LIN {X 0,Y 190.635,Z 472.728,A -85,B 0,C 180,E1 -21841.367,E2 -21841.367} C_VEL
LIN {X 0,Y 190.155,Z 472.929,A -85,B 0,C 180,E1 -21843.676,E2 -21843.676} C_VEL
LIN {X 0,Y 189.683,Z 472.071,A -85,B 0,C 180,E1 -21847.835,E2 -21847.835} C_VEL
LIN {X 0,Y 189.629,Z 470.742,A -85,B 0,C 180,E1 -21850.519,E2 -21850.519} C_VEL
LIN {X 0,Y 190.011,Z 467.936,A -85,B 0,C 180,E1 -21854.047,E2 -21854.047} C_VEL
LIN {X 0,Y 190.59,Z 464.351,A -85,B 0,C 180,E1 -21857.221,E2 -21857.221} C_VEL
LIN {X 0,Y 191.538,Z 459.248,A -85,B 0,C 180,E1 -21860.606,E2 -21860.606} C_VEL
LIN {X 0,Y 192.941,Z 452.066,A -85,B 0,C 180,E1 -21864.254,E2 -21864.254} C_VEL
LIN {X 0,Y 194.673,Z 443.985,A -85,B 0,C 180,E1 -21867.417,E2 -21867.417} C_VEL
LIN {X 0,Y 196.751,Z 434.772,A -85,B 0,C 180,E1 -21870.26,E2 -21870.26} C_VEL
LIN {X 0,Y 199.045,Z 424.398,A -85,B 0,C 180,E1 -21872.786,E2 -21872.786} C_VEL
LIN {X 0,Y 201.339,Z 412.61,A -85,B 0,C 180,E1 -21875.009,E2 -21875.009} C_VEL
LIN {X 0,Y 203.246,Z 401.02,A -85,B 0,C 180,E1 -21876.705,E2 -21876.705} C_VEL
LIN {X 0,Y 205.015,Z 388.044,A -85,B 0,C 180,E1 -21878.097,E2 -21878.097} C_VEL
LIN {X 0,Y 206.329,Z 374.818,A -85,B 0,C 180,E1 -21879.087,E2 -21879.087} C_VEL
LIN {X 0,Y 207.163,Z 361.086,A -85,B 0,C 180,E1 -21879.699,E2 -21879.699} C_VEL
LIN {X 0,Y 209.379,Z 305.404,A -85,B 0,C 180,E1 -21881.576,E2 -21881.576} C_VEL
LIN {X 0,Y 204.012,Z 288.584,A -85,B 0,C 180,E1 -21882.979,E2 -21882.979} C_VEL
LIN {X 0,Y 197.083,Z 272.096,A -85,B 0,C 180,E1 -21884.701,E2 -21884.701} C_VEL
LIN {X 0,Y 192.993,Z 264.168,A -85,B 0,C 180,E1 -21885.75,E2 -21885.75} C_VEL
LIN {X 0,Y 192.766,Z 263.116,A -85,B 0,C 180,E1 -21886.145,E2 -21886.145} C_VEL
LIN {X 0,Y 192.66,Z 262.98,A -85,B 0,C 180,E1 -21889.169,E2 -21889.169} C_VEL
LIN {X 0,Y 192.599,Z 262.997,A -85,B 0,C 180,E1 -21894.206,E2 -21894.206} C_VEL
LIN {X 0,Y 192.575,Z 263.001,A -85,B 0,C 180,E1 -21898.872,E2 -21898.872} C_VEL
LIN {X 0,Y 192.571,Z 262.983,A -85,B 0,C 180,E1 -21903.195,E2 -21903.195} C_VEL
LIN {X 0,Y 192.521,Z 262.988,A -85,B 0,C 180,E1 -21908.363,E2 -21908.363} C_VEL
LIN {X 0,Y 192.467,Z 263.009,A -85,B 0,C 180,E1 -21913.102,E2 -21913.102} C_VEL
LIN {X 0,Y 192.468,Z 262.995,A -85,B 0,C 180,E1 -21916.916,E2 -21916.916} C_VEL
LIN {X 0,Y 192.528,Z 262.99,A -85,B 0,C 180,E1 -21921.655,E2 -21921.655} C_VEL
LIN {X 0,Y 192.585,Z 262.985,A -85,B 0,C 180,E1 -21926.823,E2 -21926.823} C_VEL
LIN {X 0,Y 192.604,Z 262.959,A -85,B 0,C 180,E1 -21931.693,E2 -21931.693} C_VEL
LIN {X 0,Y 192.652,Z 262.986,A -85,B 0,C 180,E1 -21936.351,E2 -21936.351} C_VEL
LIN {X 0,Y 192.694,Z 262.947,A -85,B 0,C 180,E1 -21941.501,E2 -21941.501} C_VEL
LIN {X 0,Y 192.74,Z 262.946,A -85,B 0,C 180,E1 -21945.221,E2 -21945.221} C_VEL
LIN {X 0,Y 192.95,Z 262.949,A -85,B 0,C 180,E1 -21949.576,E2 -21949.576} C_VEL
LIN {X 0,Y 192.97,Z 262.926,A -85,B 0,C 180,E1 -21953.736,E2 -21953.736} C_VEL
LIN {X 0,Y 193.236,Z 262.875,A -85,B 0,C 180,E1 -21957.924,E2 -21957.924} C_VEL
LIN {X 0,Y 193.422,Z 262.875,A -85,B 0,C 180,E1 -21960.008,E2 -21960.008} C_VEL
LIN {X 0,Y 192.939,Z 262.951,A -85,B 0,C 180,E1 -21964.186,E2 -21964.186} C_VEL
LIN {X 0,Y 193.031,Z 262.904,A -85,B 0,C 180,E1 -21968.382,E2 -21968.382} C_VEL
LIN {X 0,Y 192.803,Z 262.955,A -85,B 0,C 180,E1 -21972.641,E2 -21972.641} C_VEL
LIN {X 0,Y 192.732,Z 262.972,A -85,B 0,C 180,E1 -21976.969,E2 -21976.969} C_VEL
LIN {X 0,Y 192.6,Z 262.967,A -85,B 0,C 180,E1 -21981.409,E2 -21981.409} C_VEL
LIN {X 0,Y 192.654,Z 262.984,A -85,B 0,C 180,E1 -21984.21,E2 -21984.21} C_VEL
LIN {X 0,Y 192.621,Z 262.97,A -85,B 0,C 180,E1 -21988.87,E2 -21988.87} C_VEL
LIN {X 0,Y 192.615,Z 262.993,A -85,B 0,C 180,E1 -21993.191,E2 -21993.191} C_VEL
LIN {X 0,Y 192.561,Z 262.99,A -85,B 0,C 180,E1 -21998.358,E2 -21998.358} C_VEL
LIN {X 0,Y 192.504,Z 262.993,A -85,B 0,C 180,E1 -22003.095,E2 -22003.095} C_VEL
LIN {X 0,Y 192.505,Z 262.996,A -85,B 0,C 180,E1 -22006.909,E2 -22006.909} C_VEL
LIN {X 0,Y 192.606,Z 263.152,A -85,B 0,C 180,E1 -22011.508,E2 -22011.508} C_VEL
LIN {X 0,Y 193.472,Z 266.43,A -85,B 0,C 180,E1 -22013.217,E2 -22013.217} C_VEL
LIN {X 0,Y 197.352,Z 275.633,A -85,B 0,C 180,E1 -22014.326,E2 -22014.326} C_VEL
LIN {X 0,Y 203.854,Z 292.087,A -85,B 0,C 180,E1 -22015.975,E2 -22015.975} C_VEL
LIN {X 0,Y 207.069,Z 301.489,A -85,B 0,C 180,E1 -22016.795,E2 -22016.795} C_VEL
LIN {X 0,Y 209.011,Z 318.594,A -85,B 0,C 180,E1 -22017.718,E2 -22017.718} C_VEL
LIN {X 0,Y 208.6,Z 329.617,A -85,B 0,C 180,E1 -22018.092,E2 -22018.092} C_VEL
LIN {X 0,Y 207.75,Z 335.448,A -85,B 0,C 180,E1 -22018.209,E2 -22018.209} C_VEL
LIN {X 0,Y 201.752,Z 354.354,A -85,B 0,C 180,E1 -22018.18,E2 -22018.18} C_VEL
LIN {X 0,Y 200.903,Z 360.185,A -85,B 0,C 180,E1 -22018.303,E2 -22018.303} C_VEL
LIN {X 0,Y 199.95,Z 377.377,A -85,B 0,C 180,E1 -22018.989,E2 -22018.989} C_VEL
LIN {X 0,Y 198.707,Z 390.244,A -85,B 0,C 180,E1 -22019.878,E2 -22019.878} C_VEL
LIN {X 0,Y 196.959,Z 403.1,A -85,B 0,C 180,E1 -22021.199,E2 -22021.199} C_VEL
LIN {X 0,Y 194.713,Z 415.331,A -85,B 0,C 180,E1 -22022.887,E2 -22022.887} C_VEL
LIN {X 0,Y 192.54,Z 426.271,A -85,B 0,C 180,E1 -22024.888,E2 -22024.888} C_VEL
LIN {X 0,Y 190.296,Z 437.059,A -85,B 0,C 180,E1 -22027.429,E2 -22027.429} C_VEL
LIN {X 0,Y 188.057,Z 446.823,A -85,B 0,C 180,E1 -22030.342,E2 -22030.342} C_VEL
LIN {X 0,Y 186.11,Z 455.204,A -85,B 0,C 180,E1 -22033.544,E2 -22033.544} C_VEL
LIN {X 0,Y 184.681,Z 461.939,A -85,B 0,C 180,E1 -22036.798,E2 -22036.798} C_VEL
LIN {X 0,Y 183.755,Z 467.292,A -85,B 0,C 180,E1 -22040.086,E2 -22040.086} C_VEL
LIN {X 0,Y 183.23,Z 471.435,A -85,B 0,C 180,E1 -22043.389,E2 -22043.389} C_VEL
LIN {X 0,Y 183.008,Z 474.694,A -85,B 0,C 180,E1 -22046.943,E2 -22046.943} C_VEL
LIN {X 0,Y 183.091,Z 476.56,A -85,B 0,C 180,E1 -22049.997,E2 -22049.997} C_VEL
LIN {X 0,Y 182.987,Z 477.614,A -85,B 0,C 180,E1 -22052.932,E2 -22052.932} C_VEL
LIN {X 0,Y 183.318,Z 477.942,A -85,B 0,C 180,E1 -22056.601,E2 -22056.601} C_VEL
LIN {X 0,Y 184.259,Z 476.916,A -85,B 0,C 180,E1 -22060.991,E2 -22060.991} C_VEL
LIN {X 0,Y 185.09,Z 475.826,A -85,B 0,C 180,E1 -22063.165,E2 -22063.165} C_VEL
LIN {X 0,Y 187.406,Z 472.371,A -85,B 0,C 180,E1 -22067.455,E2 -22067.455} C_VEL
LIN {X 0,Y 189.98,Z 468.647,A -85,B 0,C 180,E1 -22070.572,E2 -22070.572} C_VEL
LIN {X 0,Y 193.063,Z 463.838,A -85,B 0,C 180,E1 -22073.601,E2 -22073.601} C_VEL
LIN {X 0,Y 196.79,Z 457.336,A -85,B 0,C 180,E1 -22076.756,E2 -22076.756} C_VEL
LIN {X 0,Y 200.573,Z 450.34,A -85,B 0,C 180,E1 -22079.373,E2 -22079.373} C_VEL
LIN {X 0,Y 204.416,Z 442.725,A -85,B 0,C 180,E1 -22081.618,E2 -22081.618} C_VEL
LIN {X 0,Y 208.897,Z 432.451,A -85,B 0,C 180,E1 -22084.005,E2 -22084.005} C_VEL
LIN {X 0,Y 212.902,Z 422.02,A -85,B 0,C 180,E1 -22085.865,E2 -22085.865} C_VEL
LIN {X 0,Y 216.718,Z 410.439,A -85,B 0,C 180,E1 -22087.444,E2 -22087.444} C_VEL
LIN {X 0,Y 219.89,Z 398.149,A -85,B 0,C 180,E1 -22088.696,E2 -22088.696} C_VEL
LIN {X 0,Y 222.444,Z 385.35,A -85,B 0,C 180,E1 -22089.619,E2 -22089.619} C_VEL
LIN {X 0,Y 224.08,Z 373.434,A -85,B 0,C 180,E1 -22090.191,E2 -22090.191} C_VEL
LIN {X 0,Y 226.848,Z 330.995,A -85,B 0,C 180,E1 -22091.536,E2 -22091.536} C_VEL
LIN {X 0,Y 221.284,Z 318.167,A -85,B 0,C 180,E1 -22093.904,E2 -22093.904} C_VEL
LIN {X 0,Y 216.569,Z 309.026,A -85,B 0,C 180,E1 -22096.018,E2 -22096.018} C_VEL
LIN {X 0,Y 211.954,Z 300.85,A -85,B 0,C 180,E1 -22098.281,E2 -22098.281} C_VEL
LIN {X 0,Y 207.464,Z 293.64,A -85,B 0,C 180,E1 -22100.692,E2 -22100.692} C_VEL
LIN {X 0,Y 203.953,Z 288.361,A -85,B 0,C 180,E1 -22102.755,E2 -22102.755} C_VEL
LIN {X 0,Y 200.028,Z 282.686,A -85,B 0,C 180,E1 -22105.348,E2 -22105.348} C_VEL
LIN {X 0,Y 197.248,Z 278.883,A -85,B 0,C 180,E1 -22107.418,E2 -22107.418} C_VEL
LIN {X 0,Y 196.06,Z 277.275,A -85,B 0,C 180,E1 -22108.374,E2 -22108.374} C_VEL
LIN {X 0,Y 191.461,Z 271.579,A -85,B 0,C 180,E1 -22112.606,E2 -22112.606} C_VEL
LIN {X 0,Y 189.353,Z 269.308,A -85,B 0,C 180,E1 -22115.019,E2 -22115.019} C_VEL
LIN {X 0,Y 186.616,Z 266.825,A -85,B 0,C 180,E1 -22118.884,E2 -22118.884} C_VEL
LIN {X 0,Y 185.692,Z 264.067,A -85,B 0,C 180,E1 -22121.68,E2 -22121.68} C_VEL
LIN {X 0,Y 185.709,Z 263.839,A -85,B 0,C 180,E1 -22126.868,E2 -22126.868} C_VEL
LIN {X 0,Y 185.966,Z 263.808,A -85,B 0,C 180,E1 -22131.297,E2 -22131.297} C_VEL
LIN {X 0,Y 186.22,Z 263.783,A -85,B 0,C 180,E1 -22138.64,E2 -22138.64} C_VEL
LIN {X 0,Y 186.451,Z 264.522,A -85,B 0,C 180,E1 -22139.587,E2 -22139.587} C_VEL
LIN {X 0,Y 187.644,Z 267.293,A -85,B 0,C 180,E1 -22141.87,E2 -22141.87} C_VEL
LIN {X 0,Y 189.656,Z 269.253,A -85,B 0,C 180,E1 -22144.535,E2 -22144.535} C_VEL
LIN {X 0,Y 191.222,Z 269.974,A -85,B 0,C 180,E1 -22146.203,E2 -22146.203} C_VEL
LIN {X 0,Y 192.946,Z 273.232,A -85,B 0,C 180,E1 -22148.106,E2 -22148.106} C_VEL
LIN {X 0,Y 195.868,Z 275.837,A -85,B 0,C 180,E1 -22150.588,E2 -22150.588} C_VEL
LIN {X 0,Y 197.701,Z 278.85,A -85,B 0,C 180,E1 -22152.111,E2 -22152.111} C_VEL
LIN {X 0,Y 200.141,Z 281.243,A -85,B 0,C 180,E1 -22153.832,E2 -22153.832} C_VEL
LIN {X 0,Y 202.623,Z 284.781,A -85,B 0,C 180,E1 -22155.524,E2 -22155.524} C_VEL
LIN {X 0,Y 204.648,Z 287.351,A -85,B 0,C 180,E1 -22156.757,E2 -22156.757} C_VEL
LIN {X 0,Y 208.554,Z 293.119,A -85,B 0,C 180,E1 -22159.003,E2 -22159.003} C_VEL
LIN {X 0,Y 212.182,Z 298.667,A -85,B 0,C 180,E1 -22160.912,E2 -22160.912} C_VEL
LIN {X 0,Y 216.71,Z 306.479,A -85,B 0,C 180,E1 -22163.126,E2 -22163.126} C_VEL
LIN {X 0,Y 222.132,Z 316.635,A -85,B 0,C 180,E1 -22165.524,E2 -22165.524} C_VEL
LIN {X 0,Y 226.91,Z 327.095,A -85,B 0,C 180,E1 -22167.525,E2 -22167.525} C_VEL
LIN {X 0,Y 227.115,Z 328.361,A -85,B 0,C 180,E1 -22167.648,E2 -22167.648} C_VEL
LIN {X 0,Y 224.094,Z 370.541,A -85,B 0,C 180,E1 -22168.942,E2 -22168.942} C_VEL
LIN {X 0,Y 222.167,Z 384.168,A -85,B 0,C 180,E1 -22169.671,E2 -22169.671} C_VEL
LIN {X 0,Y 219.639,Z 396.507,A -85,B 0,C 180,E1 -22170.658,E2 -22170.658} C_VEL
LIN {X 0,Y 216.38,Z 408.688,A -85,B 0,C 180,E1 -22172.017,E2 -22172.017} C_VEL
LIN {X 0,Y 212.434,Z 420.621,A -85,B 0,C 180,E1 -22173.782,E2 -22173.782} C_VEL
LIN {X 0,Y 208.139,Z 431.357,A -85,B 0,C 180,E1 -22175.873,E2 -22175.873} C_VEL
LIN {X 0,Y 203.857,Z 440.688,A -85,B 0,C 180,E1 -22178.214,E2 -22178.214} C_VEL
LIN {X 0,Y 199.668,Z 448.809,A -85,B 0,C 180,E1 -22180.826,E2 -22180.826} C_VEL
LIN {X 0,Y 195.4,Z 456.305,A -85,B 0,C 180,E1 -22184.005,E2 -22184.005} C_VEL
LIN {X 0,Y 192.082,Z 461.718,A -85,B 0,C 180,E1 -22187.021,E2 -22187.021} C_VEL
LIN {X 0,Y 188.779,Z 466.675,A -85,B 0,C 180,E1 -22190.741,E2 -22190.741} C_VEL
LIN {X 0,Y 187.16,Z 468.937,A -85,B 0,C 180,E1 -22193.077,E2 -22193.077} C_VEL
LIN {X 0,Y 185.294,Z 471.326,A -85,B 0,C 180,E1 -22196.538,E2 -22196.538} C_VEL
LIN {X 0,Y 183.841,Z 472.706,A -85,B 0,C 180,E1 -22200.204,E2 -22200.204} C_VEL
LIN {X 0,Y 183.243,Z 473.013,A -85,B 0,C 180,E1 -22202.601,E2 -22202.601} C_VEL
LIN {X 0,Y 182.809,Z 472.866,A -85,B 0,C 180,E1 -22204.987,E2 -22204.987} C_VEL
LIN {X 0,Y 182.6,Z 472.195,A -85,B 0,C 180,E1 -22207.449,E2 -22207.449} C_VEL
LIN {X 0,Y 182.535,Z 471.16,A -85,B 0,C 180,E1 -22209.729,E2 -22209.729} C_VEL
LIN {X 0,Y 182.868,Z 468.141,A -85,B 0,C 180,E1 -22213.867,E2 -22213.867} C_VEL
LIN {X 0,Y 183.645,Z 463.691,A -85,B 0,C 180,E1 -22217.853,E2 -22217.853} C_VEL
LIN {X 0,Y 184.693,Z 458.053,A -85,B 0,C 180,E1 -22221.561,E2 -22221.561} C_VEL
LIN {X 0,Y 186.205,Z 450.909,A -85,B 0,C 180,E1 -22225.132,E2 -22225.132} C_VEL
LIN {X 0,Y 188.184,Z 442.509,A -85,B 0,C 180,E1 -22228.398,E2 -22228.398} C_VEL
LIN {X 0,Y 189.981,Z 434.432,A -85,B 0,C 180,E1 -22230.919,E2 -22230.919} C_VEL
LIN {X 0,Y 192.278,Z 424.458,A -85,B 0,C 180,E1 -22233.408,E2 -22233.408} C_VEL
LIN {X 0,Y 194.659,Z 412.658,A -85,B 0,C 180,E1 -22235.701,E2 -22235.701} C_VEL
LIN {X 0,Y 196.636,Z 401.052,A -85,B 0,C 180,E1 -22237.447,E2 -22237.447} C_VEL
LIN {X 0,Y 198.429,Z 388.419,A -85,B 0,C 180,E1 -22238.845,E2 -22238.845} C_VEL
LIN {X 0,Y 199.788,Z 375.342,A -85,B 0,C 180,E1 -22239.859,E2 -22239.859} C_VEL
LIN {X 0,Y 200.618,Z 362.401,A -85,B 0,C 180,E1 -22240.476,E2 -22240.476} C_VEL
LIN {X 0,Y 203.003,Z 306.497,A -85,B 0,C 180,E1 -22242.401,E2 -22242.401} C_VEL
LIN {X 0,Y 197.437,Z 289.796,A -85,B 0,C 180,E1 -22243.902,E2 -22243.902} C_VEL
LIN {X 0,Y 191.196,Z 275.061,A -85,B 0,C 180,E1 -22245.538,E2 -22245.538} C_VEL
LIN {X 0,Y 185.917,Z 264.916,A -85,B 0,C 180,E1 -22246.984,E2 -22246.984} C_VEL
LIN {X 0,Y 185.69,Z 263.966,A -85,B 0,C 180,E1 -22247.415,E2 -22247.415} C_VEL
LIN {X 0,Y 185.534,Z 263.865,A -85,B 0,C 180,E1 -22252.263,E2 -22252.263} C_VEL
LIN {X 0,Y 185.475,Z 263.871,A -85,B 0,C 180,E1 -22257.049,E2 -22257.049} C_VEL
LIN {X 0,Y 185.519,Z 263.88,A -85,B 0,C 180,E1 -22259.507,E2 -22259.507} C_VEL
LIN {X 0,Y 185.475,Z 263.876,A -85,B 0,C 180,E1 -22264.641,E2 -22264.641} C_VEL
LIN {X 0,Y 185.479,Z 263.877,A -85,B 0,C 180,E1 -22267.323,E2 -22267.323} C_VEL
LIN {X 0,Y 185.441,Z 263.863,A -85,B 0,C 180,E1 -22270.729,E2 -22270.729} C_VEL
LIN {X 0,Y 185.439,Z 263.878,A -85,B 0,C 180,E1 -22276.066,E2 -22276.066} C_VEL
LIN {X 0,Y 185.441,Z 263.856,A -85,B 0,C 180,E1 -22279.901,E2 -22279.901} C_VEL
LIN {X 0,Y 185.489,Z 263.874,A -85,B 0,C 180,E1 -22282.724,E2 -22282.724} C_VEL
LIN {X 0,Y 185.521,Z 263.851,A -85,B 0,C 180,E1 -22287.982,E2 -22287.982} C_VEL
LIN {X 0,Y 185.485,Z 263.861,A -85,B 0,C 180,E1 -22292.966,E2 -22292.966} C_VEL
LIN {X 0,Y 185.543,Z 263.869,A -85,B 0,C 180,E1 -22297.752,E2 -22297.752} C_VEL
LIN {X 0,Y 185.653,Z 263.814,A -85,B 0,C 180,E1 -22302.381,E2 -22302.381} C_VEL
LIN {X 0,Y 185.721,Z 263.837,A -85,B 0,C 180,E1 -22306.886,E2 -22306.886} C_VEL
LIN {X 0,Y 185.978,Z 263.817,A -85,B 0,C 180,E1 -22311.315,E2 -22311.315} C_VEL
LIN {X 0,Y 186.182,Z 263.751,A -85,B 0,C 180,E1 -22317.845,E2 -22317.845} C_VEL
LIN {X 0,Y 186.388,Z 263.751,A -85,B 0,C 180,E1 -22320.008,E2 -22320.008} C_VEL
LIN {X 0,Y 185.888,Z 263.828,A -85,B 0,C 180,E1 -22324.345,E2 -22324.345} C_VEL
LIN {X 0,Y 185.982,Z 263.778,A -85,B 0,C 180,E1 -22328.702,E2 -22328.702} C_VEL
LIN {X 0,Y 185.73,Z 263.84,A -85,B 0,C 180,E1 -22333.131,E2 -22333.131} C_VEL
LIN {X 0,Y 185.669,Z 263.848,A -85,B 0,C 180,E1 -22337.635,E2 -22337.635} C_VEL
LIN {X 0,Y 185.571,Z 263.848,A -85,B 0,C 180,E1 -22342.263,E2 -22342.263} C_VEL
LIN {X 0,Y 185.596,Z 263.865,A -85,B 0,C 180,E1 -22344.652,E2 -22344.652} C_VEL
LIN {X 0,Y 185.564,Z 263.846,A -85,B 0,C 180,E1 -22349.504,E2 -22349.504} C_VEL
LIN {X 0,Y 185.517,Z 263.872,A -85,B 0,C 180,E1 -22354.637,E2 -22354.637} C_VEL
LIN {X 0,Y 185.52,Z 263.859,A -85,B 0,C 180,E1 -22357.318,E2 -22357.318} C_VEL
LIN {X 0,Y 185.481,Z 263.878,A -85,B 0,C 180,E1 -22360.724,E2 -22360.724} C_VEL
LIN {X 0,Y 185.476,Z 263.875,A -85,B 0,C 180,E1 -22366.059,E2 -22366.059} C_VEL
LIN {X 0,Y 185.551,Z 264.047,A -85,B 0,C 180,E1 -22370.73,E2 -22370.73} C_VEL
LIN {X 0,Y 186.107,Z 266.268,A -85,B 0,C 180,E1 -22371.904,E2 -22371.904} C_VEL
LIN {X 0,Y 189.248,Z 273.203,A -85,B 0,C 180,E1 -22372.877,E2 -22372.877} C_VEL
LIN {X 0,Y 197.263,Z 292.951,A -85,B 0,C 180,E1 -22375.039,E2 -22375.039} C_VEL
LIN {X 0,Y 200.853,Z 303.693,A -85,B 0,C 180,E1 -22376.015,E2 -22376.015} C_VEL
LIN {X 0,Y 202.601,Z 318.627,A -85,B 0,C 180,E1 -22376.866,E2 -22376.866} C_VEL
LIN {X 0,Y 200.903,Z 360.185,A -85,B 0,C 180,E1 -22378.303,E2 -22378.303} C_VEL
LIN {X 0,Y 200.027,Z 366.019,A -85,B 0,C 180,E1 -22378.418,E2 -22378.418} C_VEL
LIN {X 0,Y 196.863,Z 375.429,A -85,B 0,C 180,E1 -22378.47,E2 -22378.47} C_VEL
LIN {X 0,Y 193.445,Z 384.704,A -85,B 0,C 180,E1 -22378.682,E2 -22378.682} C_VEL
LIN {X 0,Y 192.18,Z 390.322,A -85,B 0,C 180,E1 -22379.067,E2 -22379.067} C_VEL
LIN {X 0,Y 190.394,Z 403.014,A -85,B 0,C 180,E1 -22380.412,E2 -22380.412} C_VEL
LIN {X 0,Y 188.063,Z 415.24,A -85,B 0,C 180,E1 -22382.148,E2 -22382.148} C_VEL
LIN {X 0,Y 185.817,Z 426.18,A -85,B 0,C 180,E1 -22384.214,E2 -22384.214} C_VEL
LIN {X 0,Y 183.781,Z 435.51,A -85,B 0,C 180,E1 -22386.442,E2 -22386.442} C_VEL
LIN {X 0,Y 181.81,Z 444.296,A -85,B 0,C 180,E1 -22389.046,E2 -22389.046} C_VEL
LIN {X 0,Y 179.584,Z 453.207,A -85,B 0,C 180,E1 -22392.341,E2 -22392.341} C_VEL
LIN {X 0,Y 177.91,Z 460.308,A -85,B 0,C 180,E1 -22395.703,E2 -22395.703} C_VEL
LIN {X 0,Y 176.724,Z 466.788,A -85,B 0,C 180,E1 -22399.687,E2 -22399.687} C_VEL
LIN {X 0,Y 176.157,Z 471.025,A -85,B 0,C 180,E1 -22403.122,E2 -22403.122} C_VEL
LIN {X 0,Y 175.931,Z 474.661,A -85,B 0,C 180,E1 -22407.192,E2 -22407.192} C_VEL
LIN {X 0,Y 176.002,Z 476.321,A -85,B 0,C 180,E1 -22409.996,E2 -22409.996} C_VEL
LIN {X 0,Y 175.913,Z 477.368,A -85,B 0,C 180,E1 -22412.685,E2 -22412.685} C_VEL
LIN {X 0,Y 176.258,Z 477.863,A -85,B 0,C 180,E1 -22416.867,E2 -22416.867} C_VEL
LIN {X 0,Y 177.278,Z 476.916,A -85,B 0,C 180,E1 -22421.429,E2 -22421.429} C_VEL
LIN {X 0,Y 178.156,Z 475.878,A -85,B 0,C 180,E1 -22423.688,E2 -22423.688} C_VEL
LIN {X 0,Y 179.276,Z 474.423,A -85,B 0,C 180,E1 -22425.923,E2 -22425.923} C_VEL
LIN {X 0,Y 181.482,Z 471.461,A -85,B 0,C 180,E1 -22429.214,E2 -22429.214} C_VEL
LIN {X 0,Y 184.391,Z 467.476,A -85,B 0,C 180,E1 -22432.401,E2 -22432.401} C_VEL
LIN {X 0,Y 187.769,Z 462.379,A -85,B 0,C 180,E1 -22435.491,E2 -22435.491} C_VEL
LIN {X 0,Y 192.243,Z 454.783,A -85,B 0,C 180,E1 -22438.969,E2 -22438.969} C_VEL
LIN {X 0,Y 196.803,Z 446.623,A -85,B 0,C 180,E1 -22441.781,E2 -22441.781} C_VEL
LIN {X 0,Y 200.932,Z 438.3,A -85,B 0,C 180,E1 -22444.026,E2 -22444.026} C_VEL
LIN {X 0,Y 205.369,Z 428.071,A -85,B 0,C 180,E1 -22446.175,E2 -22446.175} C_VEL
LIN {X 0,Y 209.708,Z 416.577,A -85,B 0,C 180,E1 -22448.006,E2 -22448.006} C_VEL
LIN {X 0,Y 213.214,Z 405.252,A -85,B 0,C 180,E1 -22449.38,E2 -22449.38} C_VEL
LIN {X 0,Y 216.322,Z 392.347,A -85,B 0,C 180,E1 -22450.52,E2 -22450.52} C_VEL
LIN {X 0,Y 218.635,Z 379.17,A -85,B 0,C 180,E1 -22451.319,E2 -22451.319} C_VEL
LIN {X 0,Y 220.099,Z 364.62,A -85,B 0,C 180,E1 -22451.85,E2 -22451.85} C_VEL
LIN {X 0,Y 222.129,Z 333.652,A -85,B 0,C 180,E1 -22452.822,E2 -22452.822} C_VEL
LIN {X 0,Y 216.751,Z 321.163,A -85,B 0,C 180,E1 -22455.266,E2 -22455.266} C_VEL
LIN {X 0,Y 212.071,Z 312.005,A -85,B 0,C 180,E1 -22457.539,E2 -22457.539} C_VEL
LIN {X 0,Y 207.269,Z 303.49,A -85,B 0,C 180,E1 -22460.109,E2 -22460.109} C_VEL
LIN {X 0,Y 204.191,Z 298.619,A -85,B 0,C 180,E1 -22461.887,E2 -22461.887} C_VEL
LIN {X 0,Y 201.345,Z 294.185,A -85,B 0,C 180,E1 -22463.666,E2 -22463.666} C_VEL
LIN {X 0,Y 197.951,Z 289.004,A -85,B 0,C 180,E1 -22466.063,E2 -22466.063} C_VEL
LIN {X 0,Y 195.125,Z 284.978,A -85,B 0,C 180,E1 -22468.281,E2 -22468.281} C_VEL
LIN {X 0,Y 193.375,Z 282.885,A -85,B 0,C 180,E1 -22469.758,E2 -22469.758} C_VEL
LIN {X 0,Y 189.268,Z 277.383,A -85,B 0,C 180,E1 -22473.976,E2 -22473.976} C_VEL
LIN {X 0,Y 187.407,Z 275.728,A -85,B 0,C 180,E1 -22476.271,E2 -22476.271} C_VEL
LIN {X 0,Y 185.148,Z 273.224,A -85,B 0,C 180,E1 -22479.871,E2 -22479.871} C_VEL
LIN {X 0,Y 184.243,Z 270.842,A -85,B 0,C 180,E1 -22482.224,E2 -22482.224} C_VEL
LIN {X 0,Y 182.763,Z 270.153,A -85,B 0,C 180,E1 -22491.144,E2 -22491.144} C_VEL
LIN {X 0,Y 185.081,Z 270.999,A -85,B 0,C 180,E1 -22498.768,E2 -22498.768} C_VEL
LIN {X 0,Y 186.442,Z 274.174,A -85,B 0,C 180,E1 -22501.477,E2 -22501.477} C_VEL
LIN {X 0,Y 188.484,Z 276.202,A -85,B 0,C 180,E1 -22504.268,E2 -22504.268} C_VEL
LIN {X 0,Y 189.786,Z 277.011,A -85,B 0,C 180,E1 -22505.726,E2 -22505.726} C_VEL
LIN {X 0,Y 191.629,Z 280.228,A -85,B 0,C 180,E1 -22507.807,E2 -22507.807} C_VEL
LIN {X 0,Y 194.015,Z 282.428,A -85,B 0,C 180,E1 -22509.911,E2 -22509.911} C_VEL
LIN {X 0,Y 196.027,Z 285.561,A -85,B 0,C 180,E1 -22511.626,E2 -22511.626} C_VEL
LIN {X 0,Y 198.207,Z 287.908,A -85,B 0,C 180,E1 -22513.235,E2 -22513.235} C_VEL
LIN {X 0,Y 201.233,Z 291.945,A -85,B 0,C 180,E1 -22515.332,E2 -22515.332} C_VEL
LIN {X 0,Y 205.848,Z 298.959,A -85,B 0,C 180,E1 -22518.166,E2 -22518.166} C_VEL
LIN {X 0,Y 210.427,Z 306.18,A -85,B 0,C 180,E1 -22520.664,E2 -22520.664} C_VEL
LIN {X 0,Y 216.676,Z 317.888,A -85,B 0,C 180,E1 -22523.761,E2 -22523.761} C_VEL
LIN {X 0,Y 221.348,Z 327.813,A -85,B 0,C 180,E1 -22525.863,E2 -22525.863} C_VEL
LIN {X 0,Y 222.395,Z 330.231,A -85,B 0,C 180,E1 -22526.319,E2 -22526.319} C_VEL
LIN {X 0,Y 219.392,Z 370.665,A -85,B 0,C 180,E1 -22527.576,E2 -22527.576} C_VEL
LIN {X 0,Y 217.332,Z 384.588,A -85,B 0,C 180,E1 -22528.324,E2 -22528.324} C_VEL
LIN {X 0,Y 214.723,Z 396.785,A -85,B 0,C 180,E1 -22529.314,E2 -22529.314} C_VEL
LIN {X 0,Y 211.378,Z 408.758,A -85,B 0,C 180,E1 -22530.656,E2 -22530.656} C_VEL
LIN {X 0,Y 207.695,Z 419.493,A -85,B 0,C 180,E1 -22532.232,E2 -22532.232} C_VEL
LIN {X 0,Y 203.677,Z 429.414,A -85,B 0,C 180,E1 -22534.099,E2 -22534.099} C_VEL
LIN {X 0,Y 199.297,Z 438.751,A -85,B 0,C 180,E1 -22536.356,E2 -22536.356} C_VEL
LIN {X 0,Y 194.632,Z 447.474,A -85,B 0,C 180,E1 -22539.079,E2 -22539.079} C_VEL
LIN {X 0,Y 191.231,Z 453.329,A -85,B 0,C 180,E1 -22541.403,E2 -22541.403} C_VEL
LIN {X 0,Y 187.314,Z 459.543,A -85,B 0,C 180,E1 -22544.536,E2 -22544.536} C_VEL
LIN {X 0,Y 183.778,Z 464.704,A -85,B 0,C 180,E1 -22547.997,E2 -22547.997} C_VEL
LIN {X 0,Y 180.934,Z 468.545,A -85,B 0,C 180,E1 -22551.58,E2 -22551.58} C_VEL
LIN {X 0,Y 178.494,Z 471.426,A -85,B 0,C 180,E1 -22555.758,E2 -22555.758} C_VEL
LIN {X 0,Y 177.125,Z 472.683,A -85,B 0,C 180,E1 -22558.952,E2 -22558.952} C_VEL
LIN {X 0,Y 176.395,Z 473.077,A -85,B 0,C 180,E1 -22561.442,E2 -22561.442} C_VEL
LIN {X 0,Y 175.854,Z 473.036,A -85,B 0,C 180,E1 -22563.925,E2 -22563.925} C_VEL
LIN {X 0,Y 175.519,Z 472.318,A -85,B 0,C 180,E1 -22567.037,E2 -22567.037} C_VEL
LIN {X 0,Y 175.491,Z 470.146,A -85,B 0,C 180,E1 -22571.318,E2 -22571.318} C_VEL
LIN {X 0,Y 175.938,Z 467.136,A -85,B 0,C 180,E1 -22574.955,E2 -22574.955} C_VEL
LIN {X 0,Y 176.72,Z 463.019,A -85,B 0,C 180,E1 -22578.534,E2 -22578.534} C_VEL
LIN {X 0,Y 177.856,Z 457.089,A -85,B 0,C 180,E1 -22582.391,E2 -22582.391} C_VEL
LIN {X 0,Y 179.489,Z 449.699,A -85,B 0,C 180,E1 -22586.074,E2 -22586.074} C_VEL
LIN {X 0,Y 181.29,Z 442.557,A -85,B 0,C 180,E1 -22588.893,E2 -22588.893} C_VEL
LIN {X 0,Y 183.364,Z 433.669,A -85,B 0,C 180,E1 -22591.738,E2 -22591.738} C_VEL
LIN {X 0,Y 185.776,Z 423.283,A -85,B 0,C 180,E1 -22594.343,E2 -22594.343} C_VEL
LIN {X 0,Y 188.016,Z 412.663,A -85,B 0,C 180,E1 -22596.442,E2 -22596.442} C_VEL
LIN {X 0,Y 190.08,Z 401.027,A -85,B 0,C 180,E1 -22598.241,E2 -22598.241} C_VEL
LIN {X 0,Y 191.868,Z 388.79,A -85,B 0,C 180,E1 -22599.638,E2 -22599.638} C_VEL
LIN {X 0,Y 193.351,Z 375.062,A -85,B 0,C 180,E1 -22600.731,E2 -22600.731} C_VEL
LIN {X 0,Y 194.247,Z 361.205,A -85,B 0,C 180,E1 -22601.385,E2 -22601.385} C_VEL
LIN {X 0,Y 196.538,Z 307.784,A -85,B 0,C 180,E1 -22603.286,E2 -22603.286} C_VEL
LIN {X 0,Y 191.42,Z 292.329,A -85,B 0,C 180,E1 -22604.747,E2 -22604.747} C_VEL
LIN {X 0,Y 185.547,Z 278.381,A -85,B 0,C 180,E1 -22606.377,E2 -22606.377} C_VEL
LIN {X 0,Y 179.953,Z 268.081,A -85,B 0,C 180,E1 -22607.914,E2 -22607.914} C_VEL
LIN {X 0,Y 178.735,Z 265.425,A -85,B 0,C 180,E1 -22608.409,E2 -22608.409} C_VEL
LIN {X 0,Y 178.607,Z 264.782,A -85,B 0,C 180,E1 -22608.923,E2 -22608.923} C_VEL
LIN {X 0,Y 178.479,Z 264.749,A -85,B 0,C 180,E1 -22615.111,E2 -22615.111} C_VEL
LIN {X 0,Y 178.436,Z 264.752,A -85,B 0,C 180,E1 -22620.803,E2 -22620.803} C_VEL
LIN {X 0,Y 178.46,Z 264.747,A -85,B 0,C 180,E1 -22624.226,E2 -22624.226} C_VEL
LIN {X 0,Y 178.367,Z 264.743,A -85,B 0,C 180,E1 -22629.086,E2 -22629.086} C_VEL
LIN {X 0,Y 178.375,Z 264.756,A -85,B 0,C 180,E1 -22632.056,E2 -22632.056} C_VEL
LIN {X 0,Y 178.374,Z 264.763,A -85,B 0,C 180,E1 -22635.175,E2 -22635.175} C_VEL
LIN {X 0,Y 178.382,Z 264.732,A -85,B 0,C 180,E1 -22638.472,E2 -22638.472} C_VEL
LIN {X 0,Y 178.407,Z 264.761,A -85,B 0,C 180,E1 -22643.792,E2 -22643.792} C_VEL
LIN {X 0,Y 178.474,Z 264.743,A -85,B 0,C 180,E1 -22646.556,E2 -22646.556} C_VEL
LIN {X 0,Y 178.415,Z 264.724,A -85,B 0,C 180,E1 -22651.802,E2 -22651.802} C_VEL
LIN {X 0,Y 178.461,Z 264.755,A -85,B 0,C 180,E1 -22656.819,E2 -22656.819} C_VEL
LIN {X 0,Y 178.607,Z 264.695,A -85,B 0,C 180,E1 -22661.662,E2 -22661.662} C_VEL
LIN {X 0,Y 178.647,Z 264.71,A -85,B 0,C 180,E1 -22666.357,E2 -22666.357} C_VEL
LIN {X 0,Y 178.909,Z 264.697,A -85,B 0,C 180,E1 -22670.969,E2 -22670.969} C_VEL
LIN {X 0,Y 179.129,Z 264.627,A -85,B 0,C 180,E1 -22677.76,E2 -22677.76} C_VEL
LIN {X 0,Y 179.353,Z 264.626,A -85,B 0,C 180,E1 -22680.009,E2 -22680.009} C_VEL
LIN {X 0,Y 178.837,Z 264.705,A -85,B 0,C 180,E1 -22684.516,E2 -22684.516} C_VEL
LIN {X 0,Y 178.914,Z 264.655,A -85,B 0,C 180,E1 -22689.049,E2 -22689.049} C_VEL
LIN {X 0,Y 178.657,Z 264.726,A -85,B 0,C 180,E1 -22693.661,E2 -22693.661} C_VEL
LIN {X 0,Y 178.571,Z 264.714,A -85,B 0,C 180,E1 -22699.158,E2 -22699.158} C_VEL
LIN {X 0,Y 178.534,Z 264.747,A -85,B 0,C 180,E1 -22705.117,E2 -22705.117} C_VEL
LIN {X 0,Y 178.48,Z 264.733,A -85,B 0,C 180,E1 -22710.799,E2 -22710.799} C_VEL
LIN {X 0,Y 178.503,Z 264.749,A -85,B 0,C 180,E1 -22714.222,E2 -22714.222} C_VEL
LIN {X 0,Y 178.408,Z 264.759,A -85,B 0,C 180,E1 -22719.081,E2 -22719.081} C_VEL
LIN {X 0,Y 178.414,Z 264.747,A -85,B 0,C 180,E1 -22722.05,E2 -22722.05} C_VEL
LIN {X 0,Y 178.412,Z 264.763,A -85,B 0,C 180,E1 -22725.168,E2 -22725.168} C_VEL
LIN {X 0,Y 178.459,Z 264.897,A -85,B 0,C 180,E1 -22729.806,E2 -22729.806} C_VEL
LIN {X 0,Y 178.88,Z 266.407,A -85,B 0,C 180,E1 -22730.551,E2 -22730.551} C_VEL
LIN {X 0,Y 184.608,Z 278.815,A -85,B 0,C 180,E1 -22732.303,E2 -22732.303} C_VEL
LIN {X 0,Y 191.769,Z 296.988,A -85,B 0,C 180,E1 -22734.346,E2 -22734.346} C_VEL
LIN {X 0,Y 194.725,Z 306.125,A -85,B 0,C 180,E1 -22735.204,E2 -22735.204} C_VEL
LIN {X 0,Y 196.197,Z 318.376,A -85,B 0,C 180,E1 -22735.941,E2 -22735.941} C_VEL
LIN {X 0,Y 193.779,Z 373.938,A -85,B 0,C 180,E1 -22737.963,E2 -22737.963} C_VEL
LIN {X 0,Y 192.518,Z 387.14,A -85,B 0,C 180,E1 -22738.803,E2 -22738.803} C_VEL
LIN {X 0,Y 192.18,Z 390.322,A -85,B 0,C 180,E1 -22739.067,E2 -22739.067} C_VEL
LIN {X 0,Y 191.327,Z 394.037,A -85,B 0,C 180,E1 -22739.368,E2 -22739.368} C_VEL
LIN {X 0,Y 188.394,Z 401.191,A -85,B 0,C 180,E1 -22739.898,E2 -22739.898} C_VEL
LIN {X 0,Y 183.126,Z 411.452,A -85,B 0,C 180,E1 -22740.868,E2 -22740.868} C_VEL
LIN {X 0,Y 181.216,Z 416.545,A -85,B 0,C 180,E1 -22741.606,E2 -22741.606} C_VEL
LIN {X 0,Y 180.821,Z 418.202,A -85,B 0,C 180,E1 -22741.904,E2 -22741.904} C_VEL
LIN {X 0,Y 178.594,Z 428.472,A -85,B 0,C 180,E1 -22744.033,E2 -22744.033} C_VEL
LIN {X 0,Y 176.366,Z 437.989,A -85,B 0,C 180,E1 -22746.513,E2 -22746.513} C_VEL
LIN {X 0,Y 174.25,Z 446.637,A -85,B 0,C 180,E1 -22749.331,E2 -22749.331} C_VEL
LIN {X 0,Y 172.14,Z 455.016,A -85,B 0,C 180,E1 -22752.779,E2 -22752.779} C_VEL
LIN {X 0,Y 170.591,Z 461.75,A -85,B 0,C 180,E1 -22756.293,E2 -22756.293} C_VEL
LIN {X 0,Y 169.473,Z 467.876,A -85,B 0,C 180,E1 -22760.448,E2 -22760.448} C_VEL
LIN {X 0,Y 168.985,Z 471.828,A -85,B 0,C 180,E1 -22764.028,E2 -22764.028} C_VEL
LIN {X 0,Y 168.839,Z 474.723,A -85,B 0,C 180,E1 -22767.611,E2 -22767.611} C_VEL
LIN {X 0,Y 168.902,Z 476.082,A -85,B 0,C 180,E1 -22769.996,E2 -22769.996} C_VEL
LIN {X 0,Y 168.838,Z 477.036,A -85,B 0,C 180,E1 -22772.382,E2 -22772.382} C_VEL
LIN {X 0,Y 169.193,Z 477.781,A -85,B 0,C 180,E1 -22777.155,E2 -22777.155} C_VEL
LIN {X 0,Y 170.317,Z 476.916,A -85,B 0,C 180,E1 -22781.903,E2 -22781.903} C_VEL
LIN {X 0,Y 172.429,Z 474.533,A -85,B 0,C 180,E1 -22786.573,E2 -22786.573} C_VEL
LIN {X 0,Y 174.795,Z 471.636,A -85,B 0,C 180,E1 -22789.98,E2 -22789.98} C_VEL
LIN {X 0,Y 177.855,Z 467.744,A -85,B 0,C 180,E1 -22793.271,E2 -22793.271} C_VEL
LIN {X 0,Y 181.38,Z 462.763,A -85,B 0,C 180,E1 -22796.457,E2 -22796.457} C_VEL
LIN {X 0,Y 185.356,Z 456.547,A -85,B 0,C 180,E1 -22799.528,E2 -22799.528} C_VEL
LIN {X 0,Y 189.998,Z 448.79,A -85,B 0,C 180,E1 -22802.431,E2 -22802.431} C_VEL
LIN {X 0,Y 195.139,Z 439.155,A -85,B 0,C 180,E1 -22805.183,E2 -22805.183} C_VEL
LIN {X 0,Y 199.758,Z 429.212,A -85,B 0,C 180,E1 -22807.361,E2 -22807.361} C_VEL
LIN {X 0,Y 203.727,Z 419.39,A -85,B 0,C 180,E1 -22809.014,E2 -22809.014} C_VEL
LIN {X 0,Y 207.853,Z 407.039,A -85,B 0,C 180,E1 -22810.604,E2 -22810.604} C_VEL
LIN {X 0,Y 211.066,Z 394.937,A -85,B 0,C 180,E1 -22811.751,E2 -22811.751} C_VEL
LIN {X 0,Y 213.626,Z 381.808,A -85,B 0,C 180,E1 -22812.606,E2 -22812.606} C_VEL
LIN {X 0,Y 215.21,Z 368.999,A -85,B 0,C 180,E1 -22813.142,E2 -22813.142} C_VEL
LIN {X 0,Y 217.448,Z 336.172,A -85,B 0,C 180,E1 -22814.197,E2 -22814.197} C_VEL
LIN {X 0,Y 212.698,Z 324.954,A -85,B 0,C 180,E1 -22816.511,E2 -22816.511} C_VEL
LIN {X 0,Y 207.354,Z 314.284,A -85,B 0,C 180,E1 -22819.35,E2 -22819.35} C_VEL
LIN {X 0,Y 202.422,Z 305.691,A -85,B 0,C 180,E1 -22822.243,E2 -22822.243} C_VEL
LIN {X 0,Y 198.763,Z 299.904,A -85,B 0,C 180,E1 -22824.65,E2 -22824.65} C_VEL
LIN {X 0,Y 195.758,Z 295.189,A -85,B 0,C 180,E1 -22826.898,E2 -22826.898} C_VEL
LIN {X 0,Y 192.404,Z 290.249,A -85,B 0,C 180,E1 -22829.726,E2 -22829.726} C_VEL
LIN {X 0,Y 187.735,Z 283.975,A -85,B 0,C 180,E1 -22834.659,E2 -22834.659} C_VEL
LIN {X 0,Y 183.993,Z 280.101,A -85,B 0,C 180,E1 -22840.304,E2 -22840.304} C_VEL
LIN {X 0,Y 183.199,Z 277.846,A -85,B 0,C 180,E1 -22842.552,E2 -22842.552} C_VEL
LIN {X 0,Y 181.855,Z 277.196,A -85,B 0,C 180,E1 -22851.099,E2 -22851.099} C_VEL
LIN {X 0,Y 183.962,Z 277.919,A -85,B 0,C 180,E1 -22858.35,E2 -22858.35} C_VEL
LIN {X 0,Y 185.053,Z 280.745,A -85,B 0,C 180,E1 -22860.74,E2 -22860.74} C_VEL
LIN {X 0,Y 187.067,Z 282.994,A -85,B 0,C 180,E1 -22863.694,E2 -22863.694} C_VEL
LIN {X 0,Y 188.29,Z 283.761,A -85,B 0,C 180,E1 -22865.129,E2 -22865.129} C_VEL
LIN {X 0,Y 190.199,Z 287.053,A -85,B 0,C 180,E1 -22867.375,E2 -22867.375} C_VEL
LIN {X 0,Y 192.2,Z 288.944,A -85,B 0,C 180,E1 -22869.218,E2 -22869.218} C_VEL
LIN {X 0,Y 194.48,Z 292.407,A -85,B 0,C 180,E1 -22871.225,E2 -22871.225} C_VEL
LIN {X 0,Y 196.181,Z 294.344,A -85,B 0,C 180,E1 -22872.535,E2 -22872.535} C_VEL
LIN {X 0,Y 199.961,Z 299.659,A -85,B 0,C 180,E1 -22875.245,E2 -22875.245} C_VEL
LIN {X 0,Y 203.452,Z 305.209,A -85,B 0,C 180,E1 -22877.467,E2 -22877.467} C_VEL
LIN {X 0,Y 207.757,Z 312.317,A -85,B 0,C 180,E1 -22879.93,E2 -22879.93} C_VEL
LIN {X 0,Y 213.277,Z 323.088,A -85,B 0,C 180,E1 -22882.833,E2 -22882.833} C_VEL
LIN {X 0,Y 217.69,Z 332.768,A -85,B 0,C 180,E1 -22884.934,E2 -22884.934} C_VEL
LIN {X 0,Y 214.819,Z 370.651,A -85,B 0,C 180,E1 -22886.139,E2 -22886.139} C_VEL
LIN {X 0,Y 212.725,Z 384.428,A -85,B 0,C 180,E1 -22886.879,E2 -22886.879} C_VEL
LIN {X 0,Y 210.025,Z 396.677,A -85,B 0,C 180,E1 -22887.866,E2 -22887.866} C_VEL
LIN {X 0,Y 206.419,Z 409.076,A -85,B 0,C 180,E1 -22889.261,E2 -22889.261} C_VEL
LIN {X 0,Y 202.371,Z 420.337,A -85,B 0,C 180,E1 -22890.941,E2 -22890.941} C_VEL
LIN {X 0,Y 197.907,Z 430.737,A -85,B 0,C 180,E1 -22892.976,E2 -22892.976} C_VEL
LIN {X 0,Y 192.946,Z 440.633,A -85,B 0,C 180,E1 -22895.499,E2 -22895.499} C_VEL
LIN {X 0,Y 188.088,Z 449.12,A -85,B 0,C 180,E1 -22898.316,E2 -22898.316} C_VEL
LIN {X 0,Y 183.336,Z 456.573,A -85,B 0,C 180,E1 -22901.63,E2 -22901.63} C_VEL
LIN {X 0,Y 179.226,Z 462.426,A -85,B 0,C 180,E1 -22905.109,E2 -22905.109} C_VEL
LIN {X 0,Y 175.826,Z 466.865,A -85,B 0,C 180,E1 -22908.708,E2 -22908.708} C_VEL
LIN {X 0,Y 173.11,Z 470.11,A -85,B 0,C 180,E1 -22912.49,E2 -22912.49} C_VEL
LIN {X 0,Y 171.687,Z 471.582,A -85,B 0,C 180,E1 -22915.039,E2 -22915.039} C_VEL
LIN {X 0,Y 170.485,Z 472.593,A -85,B 0,C 180,E1 -22917.599,E2 -22917.599} C_VEL
LIN {X 0,Y 169.503,Z 473.16,A -85,B 0,C 180,E1 -22920.518,E2 -22920.518} C_VEL
LIN {X 0,Y 168.958,Z 473.184,A -85,B 0,C 180,E1 -22922.775,E2 -22922.775} C_VEL
LIN {X 0,Y 168.459,Z 472.443,A -85,B 0,C 180,E1 -22926.582,E2 -22926.582} C_VEL
LIN {X 0,Y 168.356,Z 470.627,A -85,B 0,C 180,E1 -22930.495,E2 -22930.495} C_VEL
LIN {X 0,Y 168.604,Z 468.55,A -85,B 0,C 180,E1 -22933.44,E2 -22933.44} C_VEL
LIN {X 0,Y 169.178,Z 465.303,A -85,B 0,C 180,E1 -22936.796,E2 -22936.796} C_VEL
LIN {X 0,Y 170.114,Z 460.595,A -85,B 0,C 180,E1 -22940.492,E2 -22940.492} C_VEL
LIN {X 0,Y 171.369,Z 454.594,A -85,B 0,C 180,E1 -22944.119,E2 -22944.119} C_VEL
LIN {X 0,Y 173.145,Z 447.067,A -85,B 0,C 180,E1 -22947.677,E2 -22947.677} C_VEL
LIN {X 0,Y 175.442,Z 438.34,A -85,B 0,C 180,E1 -22950.924,E2 -22950.924} C_VEL
LIN {X 0,Y 177.724,Z 428.969,A -85,B 0,C 180,E1 -22953.688,E2 -22953.688} C_VEL
LIN {X 0,Y 180.223,Z 418.267,A -85,B 0,C 180,E1 -22956.16,E2 -22956.16} C_VEL
LIN {X 0,Y 182.635,Z 406.373,A -85,B 0,C 180,E1 -22958.3,E2 -22958.3} C_VEL
LIN {X 0,Y 184.611,Z 394.783,A -85,B 0,C 180,E1 -22959.867,E2 -22959.867} C_VEL
LIN {X 0,Y 186.302,Z 381.493,A -85,B 0,C 180,E1 -22961.176,E2 -22961.176} C_VEL
LIN {X 0,Y 187.427,Z 368.813,A -85,B 0,C 180,E1 -22962.001,E2 -22962.001} C_VEL
LIN {X 0,Y 190.269,Z 310.306,A -85,B 0,C 180,E1 -22964.152,E2 -22964.152} C_VEL
LIN {X 0,Y 188.815,Z 304.797,A -85,B 0,C 180,E1 -22964.63,E2 -22964.63} C_VEL
LIN {X 0,Y 184.632,Z 292.69,A -85,B 0,C 180,E1 -22965.889,E2 -22965.889} C_VEL
LIN {X 0,Y 179.627,Z 281.146,A -85,B 0,C 180,E1 -22967.356,E2 -22967.356} C_VEL
LIN {X 0,Y 173.177,Z 269.335,A -85,B 0,C 180,E1 -22969.254,E2 -22969.254} C_VEL
LIN {X 0,Y 171.672,Z 266.462,A -85,B 0,C 180,E1 -22969.783,E2 -22969.783} C_VEL
LIN {X 0,Y 171.469,Z 265.676,A -85,B 0,C 180,E1 -22970.321,E2 -22970.321} C_VEL
LIN {X 0,Y 171.409,Z 265.624,A -85,B 0,C 180,E1 -22975.599,E2 -22975.599} C_VEL
LIN {X 0,Y 171.393,Z 265.631,A -85,B 0,C 180,E1 -22980.581,E2 -22980.581} C_VEL
LIN {X 0,Y 171.37,Z 265.636,A -85,B 0,C 180,E1 -22985.044,E2 -22985.044} C_VEL
LIN {X 0,Y 171.323,Z 265.621,A -85,B 0,C 180,E1 -22988.81,E2 -22988.81} C_VEL
LIN {X 0,Y 171.301,Z 265.648,A -85,B 0,C 180,E1 -22994.228,E2 -22994.228} C_VEL
LIN {X 0,Y 171.315,Z 265.61,A -85,B 0,C 180,E1 -22998.99,E2 -22998.99} C_VEL
LIN {X 0,Y 171.347,Z 265.63,A -85,B 0,C 180,E1 -23002.044,E2 -23002.044} C_VEL
LIN {X 0,Y 171.387,Z 265.635,A -85,B 0,C 180,E1 -23005.104,E2 -23005.104} C_VEL
LIN {X 0,Y 171.384,Z 265.59,A -85,B 0,C 180,E1 -23010.534,E2 -23010.534} C_VEL
LIN {X 0,Y 171.399,Z 265.635,A -85,B 0,C 180,E1 -23015.804,E2 -23015.804} C_VEL
LIN {X 0,Y 171.507,Z 265.586,A -85,B 0,C 180,E1 -23020.874,E2 -23020.874} C_VEL
LIN {X 0,Y 171.56,Z 265.585,A -85,B 0,C 180,E1 -23025.781,E2 -23025.781} C_VEL
LIN {X 0,Y 171.847,Z 265.577,A -85,B 0,C 180,E1 -23030.594,E2 -23030.594} C_VEL
LIN {X 0,Y 171.785,Z 265.541,A -85,B 0,C 180,E1 -23035.316,E2 -23035.316} C_VEL
LIN {X 0,Y 172.318,Z 265.502,A -85,B 0,C 180,E1 -23040.009,E2 -23040.009} C_VEL
LIN {X 0,Y 171.787,Z 265.582,A -85,B 0,C 180,E1 -23044.702,E2 -23044.702} C_VEL
LIN {X 0,Y 171.854,Z 265.532,A -85,B 0,C 180,E1 -23049.424,E2 -23049.424} C_VEL
LIN {X 0,Y 171.572,Z 265.61,A -85,B 0,C 180,E1 -23054.236,E2 -23054.236} C_VEL
LIN {X 0,Y 171.496,Z 265.591,A -85,B 0,C 180,E1 -23059.506,E2 -23059.506} C_VEL
LIN {X 0,Y 171.462,Z 265.627,A -85,B 0,C 180,E1 -23065.604,E2 -23065.604} C_VEL
LIN {X 0,Y 171.437,Z 265.607,A -85,B 0,C 180,E1 -23070.577,E2 -23070.577} C_VEL
LIN {X 0,Y 171.413,Z 265.623,A -85,B 0,C 180,E1 -23075.04,E2 -23075.04} C_VEL
LIN {X 0,Y 171.364,Z 265.632,A -85,B 0,C 180,E1 -23078.805,E2 -23078.805} C_VEL
LIN {X 0,Y 171.339,Z 265.636,A -85,B 0,C 180,E1 -23084.222,E2 -23084.222} C_VEL
LIN {X 0,Y 171.41,Z 265.875,A -85,B 0,C 180,E1 -23088.663,E2 -23088.663} C_VEL
LIN {X 0,Y 171.627,Z 266.802,A -85,B 0,C 180,E1 -23089.062,E2 -23089.062} C_VEL
LIN {X 0,Y 175.907,Z 275.239,A -85,B 0,C 180,E1 -23090.442,E2 -23090.442} C_VEL
LIN {X 0,Y 181.204,Z 287.423,A -85,B 0,C 180,E1 -23092.071,E2 -23092.071} C_VEL
LIN {X 0,Y 186.977,Z 302.973,A -85,B 0,C 180,E1 -23093.814,E2 -23093.814} C_VEL
LIN {X 0,Y 188.544,Z 307.841,A -85,B 0,C 180,E1 -23094.293,E2 -23094.293} C_VEL
LIN {X 0,Y 189.84,Z 320.828,A -85,B 0,C 180,E1 -23095.071,E2 -23095.071} C_VEL
LIN {X 0,Y 187.379,Z 373.869,A -85,B 0,C 180,E1 -23097.05,E2 -23097.05} C_VEL
LIN {X 0,Y 186.068,Z 387.058,A -85,B 0,C 180,E1 -23097.913,E2 -23097.913} C_VEL
LIN {X 0,Y 184.352,Z 399.836,A -85,B 0,C 180,E1 -23099.181,E2 -23099.181} C_VEL
LIN {X 0,Y 182.183,Z 411.985,A -85,B 0,C 180,E1 -23100.851,E2 -23100.851} C_VEL
LIN {X 0,Y 180.821,Z 418.202,A -85,B 0,C 180,E1 -23101.904,E2 -23101.904} C_VEL
LIN {X 0,Y 179.183,Z 423.171,A -85,B 0,C 180,E1 -23102.799,E2 -23102.799} C_VEL
LIN {X 0,Y 174.66,Z 430.823,A -85,B 0,C 180,E1 -23104.24,E2 -23104.24} C_VEL
LIN {X 0,Y 170.147,Z 438.024,A -85,B 0,C 180,E1 -23105.935,E2 -23105.935} C_VEL
LIN {X 0,Y 168.54,Z 442.22,A -85,B 0,C 180,E1 -23107.229,E2 -23107.229} C_VEL
LIN {X 0,Y 166.379,Z 450.273,A -85,B 0,C 180,E1 -23110.246,E2 -23110.246} C_VEL
LIN {X 0,Y 164.385,Z 457.906,A -85,B 0,C 180,E1 -23113.862,E2 -23113.862} C_VEL
LIN {X 0,Y 163.055,Z 464.033,A -85,B 0,C 180,E1 -23117.551,E2 -23117.551} C_VEL
LIN {X 0,Y 162.203,Z 468.858,A -85,B 0,C 180,E1 -23121.274,E2 -23121.274} C_VEL
LIN {X 0,Y 161.817,Z 472.534,A -85,B 0,C 180,E1 -23125.013,E2 -23125.013} C_VEL
LIN {X 0,Y 161.757,Z 474.77,A -85,B 0,C 180,E1 -23128.067,E2 -23128.067} C_VEL
LIN {X 0,Y 161.756,Z 476.661,A -85,B 0,C 180,E1 -23131.925,E2 -23131.925} C_VEL
LIN {X 0,Y 161.82,Z 477.445,A -85,B 0,C 180,E1 -23134.979,E2 -23134.979} C_VEL
LIN {X 0,Y 162.153,Z 477.674,A -85,B 0,C 180,E1 -23137.467,E2 -23137.467} C_VEL
LIN {X 0,Y 162.625,Z 477.498,A -85,B 0,C 180,E1 -23139.95,E2 -23139.95} C_VEL
LIN {X 0,Y 164.359,Z 475.964,A -85,B 0,C 180,E1 -23144.862,E2 -23144.862} C_VEL
LIN {X 0,Y 165.609,Z 474.628,A -85,B 0,C 180,E1 -23147.277,E2 -23147.277} C_VEL
LIN {X 0,Y 168.144,Z 471.824,A -85,B 0,C 180,E1 -23150.806,E2 -23150.806} C_VEL
LIN {X 0,Y 171.35,Z 468.029,A -85,B 0,C 180,E1 -23154.21,E2 -23154.21} C_VEL
LIN {X 0,Y 175.053,Z 463.152,A -85,B 0,C 180,E1 -23157.493,E2 -23157.493} C_VEL
LIN {X 0,Y 179.238,Z 457.05,A -85,B 0,C 180,E1 -23160.642,E2 -23160.642} C_VEL
LIN {X 0,Y 184.096,Z 449.478,A -85,B 0,C 180,E1 -23163.606,E2 -23163.606} C_VEL
LIN {X 0,Y 189.431,Z 440.006,A -85,B 0,C 180,E1 -23166.409,E2 -23166.409} C_VEL
LIN {X 0,Y 194.221,Z 430.271,A -85,B 0,C 180,E1 -23168.619,E2 -23168.619} C_VEL
LIN {X 0,Y 198.863,Z 419.393,A -85,B 0,C 180,E1 -23170.491,E2 -23170.491} C_VEL
LIN {X 0,Y 203.141,Z 407.066,A -85,B 0,C 180,E1 -23172.086,E2 -23172.086} C_VEL
LIN {X 0,Y 206.326,Z 395.57,A -85,B 0,C 180,E1 -23173.186,E2 -23173.186} C_VEL
LIN {X 0,Y 208.868,Z 383.428,A -85,B 0,C 180,E1 -23174.015,E2 -23174.015} C_VEL
LIN {X 0,Y 210.661,Z 370.132,A -85,B 0,C 180,E1 -23174.6,E2 -23174.6} C_VEL
LIN {X 0,Y 212.966,Z 338.813,A -85,B 0,C 180,E1 -23175.601,E2 -23175.601} C_VEL
LIN {X 0,Y 208.798,Z 328.874,A -85,B 0,C 180,E1 -23177.803,E2 -23177.803} C_VEL
LIN {X 0,Y 204.135,Z 319.302,A -85,B 0,C 180,E1 -23180.45,E2 -23180.45} C_VEL
LIN {X 0,Y 199.831,Z 311.53,A -85,B 0,C 180,E1 -23183.128,E2 -23183.128} C_VEL
LIN {X 0,Y 196.391,Z 305.847,A -85,B 0,C 180,E1 -23185.551,E2 -23185.551} C_VEL
LIN {X 0,Y 193.744,Z 301.5,A -85,B 0,C 180,E1 -23187.645,E2 -23187.645} C_VEL
LIN {X 0,Y 190.657,Z 296.798,A -85,B 0,C 180,E1 -23190.381,E2 -23190.381} C_VEL
LIN {X 0,Y 186.341,Z 290.701,A -85,B 0,C 180,E1 -23195.208,E2 -23195.208} C_VEL
LIN {X 0,Y 182.904,Z 287.073,A -85,B 0,C 180,E1 -23200.629,E2 -23200.629} C_VEL
LIN {X 0,Y 182.153,Z 284.842,A -85,B 0,C 180,E1 -23202.907,E2 -23202.907} C_VEL
LIN {X 0,Y 180.946,Z 284.238,A -85,B 0,C 180,E1 -23211.054,E2 -23211.054} C_VEL
LIN {X 0,Y 182.835,Z 284.996,A -85,B 0,C 180,E1 -23217.929,E2 -23217.929} C_VEL
LIN {X 0,Y 184.101,Z 288.024,A -85,B 0,C 180,E1 -23220.743,E2 -23220.743} C_VEL
LIN {X 0,Y 186.309,Z 290.162,A -85,B 0,C 180,E1 -23223.912,E2 -23223.912} C_VEL
LIN {X 0,Y 186.953,Z 290.837,A -85,B 0,C 180,E1 -23224.718,E2 -23224.718} C_VEL
LIN {X 0,Y 189.188,Z 294.307,A -85,B 0,C 180,E1 -23227.35,E2 -23227.35} C_VEL
LIN {X 0,Y 190.474,Z 295.633,A -85,B 0,C 180,E1 -23228.585,E2 -23228.585} C_VEL
LIN {X 0,Y 193.018,Z 299.319,A -85,B 0,C 180,E1 -23230.879,E2 -23230.879} C_VEL
LIN {X 0,Y 194.317,Z 300.986,A -85,B 0,C 180,E1 -23231.928,E2 -23231.928} C_VEL
LIN {X 0,Y 197.62,Z 305.72,A -85,B 0,C 180,E1 -23234.406,E2 -23234.406} C_VEL
LIN {X 0,Y 202.606,Z 313.852,A -85,B 0,C 180,E1 -23237.679,E2 -23237.679} C_VEL
LIN {X 0,Y 206.955,Z 322.07,A -85,B 0,C 180,E1 -23240.225,E2 -23240.225} C_VEL
LIN {X 0,Y 211.884,Z 332.459,A -85,B 0,C 180,E1 -23242.865,E2 -23242.865} C_VEL
LIN {X 0,Y 213.228,Z 335.986,A -85,B 0,C 180,E1 -23243.568,E2 -23243.568} C_VEL
LIN {X 0,Y 210.388,Z 370.712,A -85,B 0,C 180,E1 -23244.648,E2 -23244.648} C_VEL
LIN {X 0,Y 208.328,Z 384.019,A -85,B 0,C 180,E1 -23245.362,E2 -23245.362} C_VEL
LIN {X 0,Y 205.537,Z 396.278,A -85,B 0,C 180,E1 -23246.325,E2 -23246.325} C_VEL
LIN {X 0,Y 202.177,Z 407.688,A -85,B 0,C 180,E1 -23247.581,E2 -23247.581} C_VEL
LIN {X 0,Y 198.177,Z 418.652,A -85,B 0,C 180,E1 -23249.167,E2 -23249.167} C_VEL
LIN {X 0,Y 193.806,Z 428.748,A -85,B 0,C 180,E1 -23251.058,E2 -23251.058} C_VEL
LIN {X 0,Y 189.134,Z 438.019,A -85,B 0,C 180,E1 -23253.281,E2 -23253.281} C_VEL
LIN {X 0,Y 184.282,Z 446.377,A -85,B 0,C 180,E1 -23255.87,E2 -23255.87} C_VEL
LIN {X 0,Y 179.699,Z 453.478,A -85,B 0,C 180,E1 -23258.725,E2 -23258.725} C_VEL
LIN {X 0,Y 175.177,Z 459.839,A -85,B 0,C 180,E1 -23262.086,E2 -23262.086} C_VEL
LIN {X 0,Y 171.188,Z 464.969,A -85,B 0,C 180,E1 -23265.745,E2 -23265.745} C_VEL
LIN {X 0,Y 168.586,Z 467.947,A -85,B 0,C 180,E1 -23268.607,E2 -23268.607} C_VEL
LIN {X 0,Y 166.929,Z 469.757,A -85,B 0,C 180,E1 -23270.843,E2 -23270.843} C_VEL
LIN {X 0,Y 165.034,Z 471.625,A -85,B 0,C 180,E1 -23273.99,E2 -23273.99} C_VEL
LIN {X 0,Y 162.88,Z 473.141,A -85,B 0,C 180,E1 -23278.821,E2 -23278.821} C_VEL
LIN {X 0,Y 162.12,Z 473.333,A -85,B 0,C 180,E1 -23281.524,E2 -23281.524} C_VEL
LIN {X 0,Y 161.394,Z 472.564,A -85,B 0,C 180,E1 -23286.1,E2 -23286.1} C_VEL
LIN {X 0,Y 161.22,Z 471.11,A -85,B 0,C 180,E1 -23289.594,E2 -23289.594} C_VEL
LIN {X 0,Y 161.476,Z 468.746,A -85,B 0,C 180,E1 -23293.199,E2 -23293.199} C_VEL
LIN {X 0,Y 162.206,Z 464.675,A -85,B 0,C 180,E1 -23297.492,E2 -23297.492} C_VEL
LIN {X 0,Y 163.335,Z 459.25,A -85,B 0,C 180,E1 -23301.666,E2 -23301.666} C_VEL
LIN {X 0,Y 164.962,Z 452.337,A -85,B 0,C 180,E1 -23305.728,E2 -23305.728} C_VEL
LIN {X 0,Y 167.048,Z 444.206,A -85,B 0,C 180,E1 -23309.401,E2 -23309.401} C_VEL
LIN {X 0,Y 169.205,Z 435.888,A -85,B 0,C 180,E1 -23312.384,E2 -23312.384} C_VEL
LIN {X 0,Y 171.878,Z 425.68,A -85,B 0,C 180,E1 -23315.282,E2 -23315.282} C_VEL
LIN {X 0,Y 174.236,Z 415.584,A -85,B 0,C 180,E1 -23317.536,E2 -23317.536} C_VEL
LIN {X 0,Y 176.443,Z 404.587,A -85,B 0,C 180,E1 -23319.46,E2 -23319.46} C_VEL
LIN {X 0,Y 178.466,Z 392.474,A -85,B 0,C 180,E1 -23321.072,E2 -23321.072} C_VEL
LIN {X 0,Y 180.13,Z 379.49,A -85,B 0,C 180,E1 -23322.308,E2 -23322.308} C_VEL
LIN {X 0,Y 181.28,Z 365.875,A -85,B 0,C 180,E1 -23323.114,E2 -23323.114} C_VEL
LIN {X 0,Y 183.999,Z 311.135,A -85,B 0,C 180,E1 -23325.161,E2 -23325.161} C_VEL
LIN {X 0,Y 179.988,Z 298.698,A -85,B 0,C 180,E1 -23326.457,E2 -23326.457} C_VEL
LIN {X 0,Y 174.761,Z 285.835,A -85,B 0,C 180,E1 -23328.099,E2 -23328.099} C_VEL
LIN {X 0,Y 168.14,Z 273.698,A -85,B 0,C 180,E1 -23330.122,E2 -23330.122} C_VEL
LIN {X 0,Y 164.652,Z 267.706,A -85,B 0,C 180,E1 -23331.278,E2 -23331.278} C_VEL
LIN {X 0,Y 164.424,Z 266.782,A -85,B 0,C 180,E1 -23331.638,E2 -23331.638} C_VEL
LIN {X 0,Y 164.331,Z 266.506,A -85,B 0,C 180,E1 -23332.642,E2 -23332.642} C_VEL
LIN {X 0,Y 164.337,Z 266.502,A -85,B 0,C 180,E1 -23336.119,E2 -23336.119} C_VEL
LIN {X 0,Y 164.329,Z 266.503,A -85,B 0,C 180,E1 -23341.223,E2 -23341.223} C_VEL
LIN {X 0,Y 164.259,Z 266.522,A -85,B 0,C 180,E1 -23346.803,E2 -23346.803} C_VEL
LIN {X 0,Y 164.266,Z 266.495,A -85,B 0,C 180,E1 -23349.928,E2 -23349.928} C_VEL
LIN {X 0,Y 164.263,Z 266.523,A -85,B 0,C 180,E1 -23353.352,E2 -23353.352} C_VEL
LIN {X 0,Y 164.244,Z 266.505,A -85,B 0,C 180,E1 -23356.808,E2 -23356.808} C_VEL
LIN {X 0,Y 164.276,Z 266.49,A -85,B 0,C 180,E1 -23360.366,E2 -23360.366} C_VEL
LIN {X 0,Y 164.315,Z 266.517,A -85,B 0,C 180,E1 -23364.362,E2 -23364.362} C_VEL
LIN {X 0,Y 164.348,Z 266.469,A -85,B 0,C 180,E1 -23369.138,E2 -23369.138} C_VEL
LIN {X 0,Y 164.351,Z 266.506,A -85,B 0,C 180,E1 -23374.695,E2 -23374.695} C_VEL
LIN {X 0,Y 164.415,Z 266.477,A -85,B 0,C 180,E1 -23380.128,E2 -23380.128} C_VEL
LIN {X 0,Y 164.487,Z 266.454,A -85,B 0,C 180,E1 -23385.156,E2 -23385.156} C_VEL
LIN {X 0,Y 164.769,Z 266.46,A -85,B 0,C 180,E1 -23390.186,E2 -23390.186} C_VEL
LIN {X 0,Y 164.824,Z 266.439,A -85,B 0,C 180,E1 -23392.661,E2 -23392.661} C_VEL
LIN {X 0,Y 165.282,Z 266.376,A -85,B 0,C 180,E1 -23400.009,E2 -23400.009} C_VEL
LIN {X 0,Y 164.828,Z 266.42,A -85,B 0,C 180,E1 -23407.358,E2 -23407.358} C_VEL
LIN {X 0,Y 164.715,Z 266.428,A -85,B 0,C 180,E1 -23411.065,E2 -23411.065} C_VEL
LIN {X 0,Y 164.454,Z 266.489,A -85,B 0,C 180,E1 -23417.416,E2 -23417.416} C_VEL
LIN {X 0,Y 164.369,Z 266.488,A -85,B 0,C 180,E1 -23422.642,E2 -23422.642} C_VEL
LIN {X 0,Y 164.389,Z 266.508,A -85,B 0,C 180,E1 -23426.122,E2 -23426.122} C_VEL
LIN {X 0,Y 164.377,Z 266.49,A -85,B 0,C 180,E1 -23431.222,E2 -23431.222} C_VEL
LIN {X 0,Y 164.3,Z 266.499,A -85,B 0,C 180,E1 -23436.798,E2 -23436.798} C_VEL
LIN {X 0,Y 164.307,Z 266.519,A -85,B 0,C 180,E1 -23439.922,E2 -23439.922} C_VEL
LIN {X 0,Y 164.302,Z 266.505,A -85,B 0,C 180,E1 -23443.345,E2 -23443.345} C_VEL
LIN {X 0,Y 164.338,Z 266.684,A -85,B 0,C 180,E1 -23447.05,E2 -23447.05} C_VEL
LIN {X 0,Y 164.528,Z 267.52,A -85,B 0,C 180,E1 -23447.474,E2 -23447.474} C_VEL
LIN {X 0,Y 166.165,Z 270.494,A -85,B 0,C 180,E1 -23448.095,E2 -23448.095} C_VEL
LIN {X 0,Y 170.846,Z 279.574,A -85,B 0,C 180,E1 -23449.602,E2 -23449.602} C_VEL
LIN {X 0,Y 175.992,Z 291.758,A -85,B 0,C 180,E1 -23451.268,E2 -23451.268} C_VEL
LIN {X 0,Y 181.48,Z 306.816,A -85,B 0,C 180,E1 -23453.026,E2 -23453.026} C_VEL
LIN {X 0,Y 182.539,Z 310.5,A -85,B 0,C 180,E1 -23453.386,E2 -23453.386} C_VEL
LIN {X 0,Y 183.597,Z 321.033,A -85,B 0,C 180,E1 -23454.051,E2 -23454.051} C_VEL
LIN {X 0,Y 180.977,Z 374.511,A -85,B 0,C 180,E1 -23456.115,E2 -23456.115} C_VEL
LIN {X 0,Y 179.574,Z 387.737,A -85,B 0,C 180,E1 -23457.023,E2 -23457.023} C_VEL
LIN {X 0,Y 177.881,Z 399.749,A -85,B 0,C 180,E1 -23458.263,E2 -23458.263} C_VEL
LIN {X 0,Y 175.634,Z 411.896,A -85,B 0,C 180,E1 -23459.984,E2 -23459.984} C_VEL
LIN {X 0,Y 173.694,Z 420.864,A -85,B 0,C 180,E1 -23461.609,E2 -23461.609} C_VEL
LIN {X 0,Y 171.419,Z 430.679,A -85,B 0,C 180,E1 -23463.845,E2 -23463.845} C_VEL
LIN {X 0,Y 168.736,Z 441.298,A -85,B 0,C 180,E1 -23466.92,E2 -23466.92} C_VEL
LIN {X 0,Y 168.54,Z 442.22,A -85,B 0,C 180,E1 -23467.229,E2 -23467.229} C_VEL
LIN {X 0,Y 167.617,Z 444.943,A -85,B 0,C 180,E1 -23468.147,E2 -23468.147} C_VEL
LIN {X 0,Y 165.305,Z 448.771,A -85,B 0,C 180,E1 -23469.492,E2 -23469.492} C_VEL
LIN {X 0,Y 158.791,Z 456.649,A -85,B 0,C 180,E1 -23472.859,E2 -23472.859} C_VEL
LIN {X 0,Y 156.966,Z 459.766,A -85,B 0,C 180,E1 -23474.573,E2 -23474.573} C_VEL
LIN {X 0,Y 156.671,Z 460.75,A -85,B 0,C 180,E1 -23475.188,E2 -23475.188} C_VEL
LIN {X 0,Y 155.444,Z 466.911,A -85,B 0,C 180,E1 -23479.577,E2 -23479.577} C_VEL
LIN {X 0,Y 154.834,Z 471.047,A -85,B 0,C 180,E1 -23483.48,E2 -23483.48} C_VEL
LIN {X 0,Y 154.677,Z 474.886,A -85,B 0,C 180,E1 -23488.695,E2 -23488.695} C_VEL
LIN {X 0,Y 154.652,Z 476.635,A -85,B 0,C 180,E1 -23492.601,E2 -23492.601} C_VEL
LIN {X 0,Y 155.092,Z 477.553,A -85,B 0,C 180,E1 -23497.809,E2 -23497.809} C_VEL
LIN {X 0,Y 155.607,Z 477.446,A -85,B 0,C 180,E1 -23500.404,E2 -23500.404} C_VEL
LIN {X 0,Y 157.498,Z 476.017,A -85,B 0,C 180,E1 -23505.525,E2 -23505.525} C_VEL
LIN {X 0,Y 160.53,Z 473.042,A -85,B 0,C 180,E1 -23510.498,E2 -23510.498} C_VEL
LIN {X 0,Y 163.716,Z 469.673,A -85,B 0,C 180,E1 -23514.063,E2 -23514.063} C_VEL
LIN {X 0,Y 167.425,Z 465.27,A -85,B 0,C 180,E1 -23517.495,E2 -23517.495} C_VEL
LIN {X 0,Y 172.16,Z 459.037,A -85,B 0,C 180,E1 -23521.123,E2 -23521.123} C_VEL
LIN {X 0,Y 177.352,Z 451.46,A -85,B 0,C 180,E1 -23524.376,E2 -23524.376} C_VEL
LIN {X 0,Y 182.885,Z 442.551,A -85,B 0,C 180,E1 -23527.242,E2 -23527.242} C_VEL
LIN {X 0,Y 187.795,Z 433.411,A -85,B 0,C 180,E1 -23529.505,E2 -23529.505} C_VEL
LIN {X 0,Y 191.944,Z 424.545,A -85,B 0,C 180,E1 -23531.224,E2 -23531.224} C_VEL
LIN {X 0,Y 196.337,Z 413.637,A -85,B 0,C 180,E1 -23532.848,E2 -23532.848} C_VEL
LIN {X 0,Y 200.281,Z 401.525,A -85,B 0,C 180,E1 -23534.216,E2 -23534.216} C_VEL
LIN {X 0,Y 203.492,Z 388.66,A -85,B 0,C 180,E1 -23535.262,E2 -23535.262} C_VEL
LIN {X 0,Y 205.831,Z 375.17,A -85,B 0,C 180,E1 -23535.969,E2 -23535.969} C_VEL
LIN {X 0,Y 207.73,Z 353.065,A -85,B 0,C 180,E1 -23536.724,E2 -23536.724} C_VEL
LIN {X 0,Y 208.616,Z 341.578,A -85,B 0,C 180,E1 -23537.083,E2 -23537.083} C_VEL
LIN {X 0,Y 204.835,Z 332.245,A -85,B 0,C 180,E1 -23539.256,E2 -23539.256} C_VEL
LIN {X 0,Y 199.719,Z 321.74,A -85,B 0,C 180,E1 -23542.411,E2 -23542.411} C_VEL
LIN {X 0,Y 194.947,Z 313.14,A -85,B 0,C 180,E1 -23545.799,E2 -23545.799} C_VEL
LIN {X 0,Y 191.664,Z 307.697,A -85,B 0,C 180,E1 -23548.49,E2 -23548.49} C_VEL
LIN {X 0,Y 188.651,Z 302.981,A -85,B 0,C 180,E1 -23551.325,E2 -23551.325} C_VEL
LIN {X 0,Y 184.777,Z 297.171,A -85,B 0,C 180,E1 -23556.02,E2 -23556.02} C_VEL
LIN {X 0,Y 182.009,Z 294.349,A -85,B 0,C 180,E1 -23560.53,E2 -23560.53} C_VEL
LIN {X 0,Y 181.145,Z 291.875,A -85,B 0,C 180,E1 -23563.166,E2 -23563.166} C_VEL
LIN {X 0,Y 180.038,Z 291.281,A -85,B 0,C 180,E1 -23571.008,E2 -23571.008} C_VEL
LIN {X 0,Y 181.728,Z 291.968,A -85,B 0,C 180,E1 -23577.498,E2 -23577.498} C_VEL
LIN {X 0,Y 183.152,Z 295.269,A -85,B 0,C 180,E1 -23580.747,E2 -23580.747} C_VEL
LIN {X 0,Y 185.515,Z 297.585,A -85,B 0,C 180,E1 -23584.133,E2 -23584.133} C_VEL
LIN {X 0,Y 187.751,Z 301.055,A -85,B 0,C 180,E1 -23586.874,E2 -23586.874} C_VEL
LIN {X 0,Y 188.882,Z 302.454,A -85,B 0,C 180,E1 -23588.048,E2 -23588.048} C_VEL
LIN {X 0,Y 191.605,Z 306.242,A -85,B 0,C 180,E1 -23590.559,E2 -23590.559} C_VEL
LIN {X 0,Y 195.365,Z 311.849,A -85,B 0,C 180,E1 -23593.58,E2 -23593.58} C_VEL
LIN {X 0,Y 199.822,Z 319.44,A -85,B 0,C 180,E1 -23596.707,E2 -23596.707} C_VEL
LIN {X 0,Y 203.962,Z 327.526,A -85,B 0,C 180,E1 -23599.273,E2 -23599.273} C_VEL
LIN {X 0,Y 208.453,Z 337.364,A -85,B 0,C 180,E1 -23601.825,E2 -23601.825} C_VEL
LIN {X 0,Y 208.872,Z 338.367,A -85,B 0,C 180,E1 -23602.055,E2 -23602.055} C_VEL
LIN {X 0,Y 206.071,Z 371.24,A -85,B 0,C 180,E1 -23603.102,E2 -23603.102} C_VEL
LIN {X 0,Y 203.84,Z 384.841,A -85,B 0,C 180,E1 -23603.841,E2 -23603.841} C_VEL
LIN {X 0,Y 200.76,Z 397.554,A -85,B 0,C 180,E1 -23604.876,E2 -23604.876} C_VEL
LIN {X 0,Y 196.905,Z 409.741,A -85,B 0,C 180,E1 -23606.272,E2 -23606.272} C_VEL
LIN {X 0,Y 192.777,Z 420.324,A -85,B 0,C 180,E1 -23607.87,E2 -23607.87} C_VEL
LIN {X 0,Y 187.683,Z 431.206,A -85,B 0,C 180,E1 -23610.023,E2 -23610.023} C_VEL
LIN {X 0,Y 182.097,Z 441.371,A -85,B 0,C 180,E1 -23612.694,E2 -23612.694} C_VEL
LIN {X 0,Y 176.918,Z 449.475,A -85,B 0,C 180,E1 -23615.483,E2 -23615.483} C_VEL
LIN {X 0,Y 171.626,Z 456.893,A -85,B 0,C 180,E1 -23618.925,E2 -23618.925} C_VEL
LIN {X 0,Y 167.512,Z 462.119,A -85,B 0,C 180,E1 -23622.151,E2 -23622.151} C_VEL
LIN {X 0,Y 163.101,Z 467.167,A -85,B 0,C 180,E1 -23626.42,E2 -23626.42} C_VEL
LIN {X 0,Y 160.908,Z 469.401,A -85,B 0,C 180,E1 -23629.074,E2 -23629.074} C_VEL
LIN {X 0,Y 158.38,Z 471.732,A -85,B 0,C 180,E1 -23632.99,E2 -23632.99} C_VEL
LIN {X 0,Y 156.275,Z 473.125,A -85,B 0,C 180,E1 -23637.344,E2 -23637.344} C_VEL
LIN {X 0,Y 155.329,Z 473.423,A -85,B 0,C 180,E1 -23640.157,E2 -23640.157} C_VEL
LIN {X 0,Y 154.668,Z 473.258,A -85,B 0,C 180,E1 -23642.979,E2 -23642.979} C_VEL
LIN {X 0,Y 154.335,Z 472.604,A -85,B 0,C 180,E1 -23645.81,E2 -23645.81} C_VEL
LIN {X 0,Y 154.124,Z 471.529,A -85,B 0,C 180,E1 -23648.609,E2 -23648.609} C_VEL
LIN {X 0,Y 154.359,Z 468.935,A -85,B 0,C 180,E1 -23652.925,E2 -23652.925} C_VEL
LIN {X 0,Y 154.965,Z 465.458,A -85,B 0,C 180,E1 -23656.898,E2 -23656.898} C_VEL
LIN {X 0,Y 155.957,Z 460.861,A -85,B 0,C 180,E1 -23660.833,E2 -23660.833} C_VEL
LIN {X 0,Y 157.381,Z 454.707,A -85,B 0,C 180,E1 -23664.88,E2 -23664.88} C_VEL
LIN {X 0,Y 159.301,Z 447.166,A -85,B 0,C 180,E1 -23668.74,E2 -23668.74} C_VEL
LIN {X 0,Y 161.718,Z 438.84,A -85,B 0,C 180,E1 -23672.088,E2 -23672.088} C_VEL
LIN {X 0,Y 164.329,Z 428.999,A -85,B 0,C 180,E1 -23675.218,E2 -23675.218} C_VEL
LIN {X 0,Y 167.001,Z 418.277,A -85,B 0,C 180,E1 -23677.865,E2 -23677.865} C_VEL
LIN {X 0,Y 169.632,Z 406.324,A -85,B 0,C 180,E1 -23680.145,E2 -23680.145} C_VEL
LIN {X 0,Y 171.75,Z 394.658,A -85,B 0,C 180,E1 -23681.81,E2 -23681.81} C_VEL
LIN {X 0,Y 173.622,Z 381.034,A -85,B 0,C 180,E1 -23683.213,E2 -23683.213} C_VEL
LIN {X 0,Y 174.833,Z 368.408,A -85,B 0,C 180,E1 -23684.052,E2 -23684.052} C_VEL
LIN {X 0,Y 177.759,Z 312.617,A -85,B 0,C 180,E1 -23686.216,E2 -23686.216} C_VEL
LIN {X 0,Y 174.278,Z 301.704,A -85,B 0,C 180,E1 -23687.416,E2 -23687.416} C_VEL
LIN {X 0,Y 169.329,Z 289.454,A -85,B 0,C 180,E1 -23689.049,E2 -23689.049} C_VEL
LIN {X 0,Y 163.212,Z 278.089,A -85,B 0,C 180,E1 -23691.024,E2 -23691.024} C_VEL
LIN {X 0,Y 158.966,Z 271.12,A -85,B 0,C 180,E1 -23692.459,E2 -23692.459} C_VEL
LIN {X 0,Y 157.435,Z 268.233,A -85,B 0,C 180,E1 -23693.125,E2 -23693.125} C_VEL
LIN {X 0,Y 157.264,Z 267.451,A -85,B 0,C 180,E1 -23693.72,E2 -23693.72} C_VEL
LIN {X 0,Y 157.267,Z 267.382,A -85,B 0,C 180,E1 -23696.676,E2 -23696.676} C_VEL
LIN {X 0,Y 157.241,Z 267.379,A -85,B 0,C 180,E1 -23702.44,E2 -23702.44} C_VEL
LIN {X 0,Y 157.237,Z 267.398,A -85,B 0,C 180,E1 -23706.454,E2 -23706.454} C_VEL
LIN {X 0,Y 157.172,Z 267.393,A -85,B 0,C 180,E1 -23712.128,E2 -23712.128} C_VEL
LIN {X 0,Y 157.174,Z 267.373,A -85,B 0,C 180,E1 -23717.893,E2 -23717.893} C_VEL
LIN {X 0,Y 157.247,Z 267.397,A -85,B 0,C 180,E1 -23723.567,E2 -23723.567} C_VEL
LIN {X 0,Y 157.266,Z 267.36,A -85,B 0,C 180,E1 -23728.119,E2 -23728.119} C_VEL
LIN {X 0,Y 157.261,Z 267.376,A -85,B 0,C 180,E1 -23733.467,E2 -23733.467} C_VEL
LIN {X 0,Y 157.358,Z 267.361,A -85,B 0,C 180,E1 -23739.714,E2 -23739.714} C_VEL
LIN {X 0,Y 157.418,Z 267.325,A -85,B 0,C 180,E1 -23744.473,E2 -23744.473} C_VEL
LIN {X 0,Y 157.691,Z 267.342,A -85,B 0,C 180,E1 -23749.741,E2 -23749.741} C_VEL
LIN {X 0,Y 157.763,Z 267.322,A -85,B 0,C 180,E1 -23752.33,E2 -23752.33} C_VEL
LIN {X 0,Y 158.244,Z 267.25,A -85,B 0,C 180,E1 -23760.01,E2 -23760.01} C_VEL
LIN {X 0,Y 157.767,Z 267.293,A -85,B 0,C 180,E1 -23767.69,E2 -23767.69} C_VEL
LIN {X 0,Y 157.646,Z 267.308,A -85,B 0,C 180,E1 -23771.233,E2 -23771.233} C_VEL
LIN {X 0,Y 157.432,Z 267.374,A -85,B 0,C 180,E1 -23775.546,E2 -23775.546} C_VEL
LIN {X 0,Y 157.327,Z 267.351,A -85,B 0,C 180,E1 -23780.948,E2 -23780.948} C_VEL
LIN {X 0,Y 157.329,Z 267.381,A -85,B 0,C 180,E1 -23786.687,E2 -23786.687} C_VEL
LIN {X 0,Y 157.288,Z 267.387,A -85,B 0,C 180,E1 -23792.435,E2 -23792.435} C_VEL
LIN {X 0,Y 157.279,Z 267.373,A -85,B 0,C 180,E1 -23796.449,E2 -23796.449} C_VEL
LIN {X 0,Y 157.21,Z 267.387,A -85,B 0,C 180,E1 -23802.122,E2 -23802.122} C_VEL
LIN {X 0,Y 157.21,Z 267.563,A -85,B 0,C 180,E1 -23805.284,E2 -23805.284} C_VEL
LIN {X 0,Y 157.538,Z 268.791,A -85,B 0,C 180,E1 -23805.831,E2 -23805.831} C_VEL
LIN {X 0,Y 159.191,Z 271.517,A -85,B 0,C 180,E1 -23806.452,E2 -23806.452} C_VEL
LIN {X 0,Y 164.045,Z 280.18,A -85,B 0,C 180,E1 -23808.117,E2 -23808.117} C_VEL
LIN {X 0,Y 169.234,Z 291.995,A -85,B 0,C 180,E1 -23809.893,E2 -23809.893} C_VEL
LIN {X 0,Y 174.929,Z 307.415,A -85,B 0,C 180,E1 -23811.82,E2 -23811.82} C_VEL
LIN {X 0,Y 176.415,Z 311.786,A -85,B 0,C 180,E1 -23812.32,E2 -23812.32} C_VEL
LIN {X 0,Y 177.354,Z 322.388,A -85,B 0,C 180,E1 -23813.003,E2 -23813.003} C_VEL
LIN {X 0,Y 174.65,Z 374.582,A -85,B 0,C 180,E1 -23815.076,E2 -23815.076} C_VEL
LIN {X 0,Y 173.215,Z 387.623,A -85,B 0,C 180,E1 -23815.998,E2 -23815.998} C_VEL
LIN {X 0,Y 171.277,Z 400.726,A -85,B 0,C 180,E1 -23817.41,E2 -23817.41} C_VEL
LIN {X 0,Y 168.733,Z 413.377,A -85,B 0,C 180,E1 -23819.317,E2 -23819.317} C_VEL
LIN {X 0,Y 166.121,Z 424.676,A -85,B 0,C 180,E1 -23821.575,E2 -23821.575} C_VEL
LIN {X 0,Y 163.882,Z 433.829,A -85,B 0,C 180,E1 -23823.92,E2 -23823.92} C_VEL
LIN {X 0,Y 161.653,Z 442.414,A -85,B 0,C 180,E1 -23826.65,E2 -23826.65} C_VEL
LIN {X 0,Y 159.3,Z 450.869,A -85,B 0,C 180,E1 -23830.002,E2 -23830.002} C_VEL
LIN {X 0,Y 157.236,Z 458.377,A -85,B 0,C 180,E1 -23833.774,E2 -23833.774} C_VEL
LIN {X 0,Y 156.671,Z 460.75,A -85,B 0,C 180,E1 -23835.188,E2 -23835.188} C_VEL
LIN {X 0,Y 155.449,Z 463.594,A -85,B 0,C 180,E1 -23837.039,E2 -23837.039} C_VEL
LIN {X 0,Y 151.82,Z 467.596,A -85,B 0,C 180,E1 -23840.141,E2 -23840.141} C_VEL
LIN {X 0,Y 148.95,Z 470.29,A -85,B 0,C 180,E1 -23842.797,E2 -23842.797} C_VEL
LIN {X 0,Y 147.706,Z 472.1,A -85,B 0,C 180,E1 -23844.941,E2 -23844.941} C_VEL
LIN {X 0,Y 147.585,Z 472.609,A -85,B 0,C 180,E1 -23845.68,E2 -23845.68} C_VEL
LIN {X 0,Y 147.649,Z 475.313,A -85,B 0,C 180,E1 -23849.996,E2 -23849.996} C_VEL
LIN {X 0,Y 147.575,Z 476.428,A -85,B 0,C 180,E1 -23852.725,E2 -23852.725} C_VEL
LIN {X 0,Y 148.046,Z 477.432,A -85,B 0,C 180,E1 -23858.183,E2 -23858.183} C_VEL
LIN {X 0,Y 149.482,Z 476.929,A -85,B 0,C 180,E1 -23863.592,E2 -23863.592} C_VEL
LIN {X 0,Y 152.059,Z 474.823,A -85,B 0,C 180,E1 -23868.872,E2 -23868.872} C_VEL
LIN {X 0,Y 156.065,Z 471.136,A -85,B 0,C 180,E1 -23873.905,E2 -23873.905} C_VEL
LIN {X 0,Y 159.828,Z 467.183,A -85,B 0,C 180,E1 -23877.493,E2 -23877.493} C_VEL
LIN {X 0,Y 164.75,Z 461.253,A -85,B 0,C 180,E1 -23881.427,E2 -23881.427} C_VEL
LIN {X 0,Y 169.777,Z 454.593,A -85,B 0,C 180,E1 -23884.689,E2 -23884.689} C_VEL
LIN {X 0,Y 175.377,Z 446.478,A -85,B 0,C 180,E1 -23887.666,E2 -23887.666} C_VEL
LIN {X 0,Y 180.31,Z 438.229,A -85,B 0,C 180,E1 -23890.02,E2 -23890.02} C_VEL
LIN {X 0,Y 185.597,Z 428.112,A -85,B 0,C 180,E1 -23892.227,E2 -23892.227} C_VEL
LIN {X 0,Y 190.709,Z 416.714,A -85,B 0,C 180,E1 -23894.068,E2 -23894.068} C_VEL
LIN {X 0,Y 194.753,Z 405.561,A -85,B 0,C 180,E1 -23895.451,E2 -23895.451} C_VEL
LIN {X 0,Y 198.117,Z 393.826,A -85,B 0,C 180,E1 -23896.525,E2 -23896.525} C_VEL
LIN {X 0,Y 200.886,Z 380.721,A -85,B 0,C 180,E1 -23897.348,E2 -23897.348} C_VEL
LIN {X 0,Y 202.649,Z 367.396,A -85,B 0,C 180,E1 -23897.878,E2 -23897.878} C_VEL
LIN {X 0,Y 204.414,Z 344.259,A -85,B 0,C 180,E1 -23898.643,E2 -23898.643} C_VEL
LIN {X 0,Y 201.201,Z 336.348,A -85,B 0,C 180,E1 -23900.623,E2 -23900.623} C_VEL
LIN {X 0,Y 196.913,Z 327.181,A -85,B 0,C 180,E1 -23903.47,E2 -23903.47} C_VEL
LIN {X 0,Y 192.556,Z 318.955,A -85,B 0,C 180,E1 -23906.798,E2 -23906.798} C_VEL
LIN {X 0,Y 189.737,Z 314.041,A -85,B 0,C 180,E1 -23909.255,E2 -23909.255} C_VEL
LIN {X 0,Y 187.033,Z 309.58,A -85,B 0,C 180,E1 -23911.958,E2 -23911.958} C_VEL
LIN {X 0,Y 183.399,Z 303.941,A -85,B 0,C 180,E1 -23916.608,E2 -23916.608} C_VEL
LIN {X 0,Y 180.882,Z 301.214,A -85,B 0,C 180,E1 -23920.983,E2 -23920.983} C_VEL
LIN {X 0,Y 180.095,Z 298.839,A -85,B 0,C 180,E1 -23923.573,E2 -23923.573} C_VEL
LIN {X 0,Y 179.127,Z 298.324,A -85,B 0,C 180,E1 -23930.962,E2 -23930.962} C_VEL
LIN {X 0,Y 180.643,Z 298.991,A -85,B 0,C 180,E1 -23937.112,E2 -23937.112} C_VEL
LIN {X 0,Y 182.178,Z 302.418,A -85,B 0,C 180,E1 -23940.697,E2 -23940.697} C_VEL
LIN {X 0,Y 184.101,Z 304.355,A -85,B 0,C 180,E1 -23943.548,E2 -23943.548} C_VEL
LIN {X 0,Y 186.406,Z 307.946,A -85,B 0,C 180,E1 -23946.486,E2 -23946.486} C_VEL
LIN {X 0,Y 187.26,Z 309.123,A -85,B 0,C 180,E1 -23947.426,E2 -23947.426} C_VEL
LIN {X 0,Y 190.493,Z 313.878,A -85,B 0,C 180,E1 -23950.523,E2 -23950.523} C_VEL
LIN {X 0,Y 193.289,Z 318.197,A -85,B 0,C 180,E1 -23952.843,E2 -23952.843} C_VEL
LIN {X 0,Y 197.58,Z 325.974,A -85,B 0,C 180,E1 -23956.036,E2 -23956.036} C_VEL
LIN {X 0,Y 201.687,Z 334.36,A -85,B 0,C 180,E1 -23958.701,E2 -23958.701} C_VEL
LIN {X 0,Y 204.688,Z 341.402,A -85,B 0,C 180,E1 -23960.522,E2 -23960.522} C_VEL
LIN {X 0,Y 202.103,Z 370.723,A -85,B 0,C 180,E1 -23961.451,E2 -23961.451} C_VEL
LIN {X 0,Y 199.982,Z 383.515,A -85,B 0,C 180,E1 -23962.114,E2 -23962.114} C_VEL
LIN {X 0,Y 196.893,Z 396.353,A -85,B 0,C 180,E1 -23963.109,E2 -23963.109} C_VEL
LIN {X 0,Y 192.995,Z 408.506,A -85,B 0,C 180,E1 -23964.45,E2 -23964.45} C_VEL
LIN {X 0,Y 188.682,Z 419.316,A -85,B 0,C 180,E1 -23966.034,E2 -23966.034} C_VEL
LIN {X 0,Y 183.365,Z 430.433,A -85,B 0,C 180,E1 -23968.18,E2 -23968.18} C_VEL
LIN {X 0,Y 177.735,Z 440.307,A -85,B 0,C 180,E1 -23970.728,E2 -23970.728} C_VEL
LIN {X 0,Y 172.543,Z 448.229,A -85,B 0,C 180,E1 -23973.391,E2 -23973.391} C_VEL
LIN {X 0,Y 167.703,Z 454.812,A -85,B 0,C 180,E1 -23976.256,E2 -23976.256} C_VEL
LIN {X 0,Y 162.353,Z 461.392,A -85,B 0,C 180,E1 -23980.099,E2 -23980.099} C_VEL
LIN {X 0,Y 157.525,Z 466.633,A -85,B 0,C 180,E1 -23984.458,E2 -23984.458} C_VEL
LIN {X 0,Y 155.051,Z 469.039,A -85,B 0,C 180,E1 -23987.17,E2 -23987.17} C_VEL
LIN {X 0,Y 151.746,Z 471.846,A -85,B 0,C 180,E1 -23991.918,E2 -23991.918} C_VEL
LIN {X 0,Y 149.783,Z 473.108,A -85,B 0,C 180,E1 -23995.738,E2 -23995.738} C_VEL
LIN {X 0,Y 148.654,Z 473.488,A -85,B 0,C 180,E1 -23998.669,E2 -23998.669} C_VEL
LIN {X 0,Y 147.815,Z 473.434,A -85,B 0,C 180,E1 -24001.616,E2 -24001.616} C_VEL
LIN {X 0,Y 147.308,Z 472.791,A -85,B 0,C 180,E1 -24004.994,E2 -24004.994} C_VEL
LIN {X 0,Y 147.027,Z 470.488,A -85,B 0,C 180,E1 -24010.456,E2 -24010.456} C_VEL
LIN {X 0,Y 147.496,Z 467.443,A -85,B 0,C 180,E1 -24014.812,E2 -24014.812} C_VEL
LIN {X 0,Y 148.348,Z 463.291,A -85,B 0,C 180,E1 -24019.081,E2 -24019.081} C_VEL
LIN {X 0,Y 149.624,Z 457.915,A -85,B 0,C 180,E1 -24023.261,E2 -24023.261} C_VEL
LIN {X 0,Y 151.345,Z 451.143,A -85,B 0,C 180,E1 -24027.343,E2 -24027.343} C_VEL
LIN {X 0,Y 153.318,Z 444.227,A -85,B 0,C 180,E1 -24030.661,E2 -24030.661} C_VEL
LIN {X 0,Y 155.713,Z 435.789,A -85,B 0,C 180,E1 -24033.916,E2 -24033.916} C_VEL
LIN {X 0,Y 158.589,Z 425.623,A -85,B 0,C 180,E1 -24037.004,E2 -24037.004} C_VEL
LIN {X 0,Y 161.185,Z 415.436,A -85,B 0,C 180,E1 -24039.414,E2 -24039.414} C_VEL
LIN {X 0,Y 163.562,Z 404.369,A -85,B 0,C 180,E1 -24041.466,E2 -24041.466} C_VEL
LIN {X 0,Y 165.672,Z 392.797,A -85,B 0,C 180,E1 -24043.093,E2 -24043.093} C_VEL
LIN {X 0,Y 167.419,Z 380.206,A -85,B 0,C 180,E1 -24044.378,E2 -24044.378} C_VEL
LIN {X 0,Y 168.65,Z 366.952,A -85,B 0,C 180,E1 -24045.234,E2 -24045.234} C_VEL
LIN {X 0,Y 171.53,Z 314.725,A -85,B 0,C 180,E1 -24047.312,E2 -24047.312} C_VEL
LIN {X 0,Y 170.844,Z 311.571,A -85,B 0,C 180,E1 -24047.608,E2 -24047.608} C_VEL
LIN {X 0,Y 167.124,Z 300.656,A -85,B 0,C 180,E1 -24048.944,E2 -24048.944} C_VEL
LIN {X 0,Y 163.406,Z 292.031,A -85,B 0,C 180,E1 -24050.229,E2 -24050.229} C_VEL
LIN {X 0,Y 157.625,Z 281.321,A -85,B 0,C 180,E1 -24052.227,E2 -24052.227} C_VEL
LIN {X 0,Y 152.079,Z 272.304,A -85,B 0,C 180,E1 -24054.264,E2 -24054.264} C_VEL
LIN {X 0,Y 150.437,Z 269.496,A -85,B 0,C 180,E1 -24054.989,E2 -24054.989} C_VEL
LIN {X 0,Y 150.223,Z 268.544,A -85,B 0,C 180,E1 -24055.436,E2 -24055.436} C_VEL
LIN {X 0,Y 150.204,Z 268.263,A -85,B 0,C 180,E1 -24057.278,E2 -24057.278} C_VEL
LIN {X 0,Y 150.182,Z 268.257,A -85,B 0,C 180,E1 -24062.635,E2 -24062.635} C_VEL
LIN {X 0,Y 150.149,Z 268.268,A -85,B 0,C 180,E1 -24067.485,E2 -24067.485} C_VEL
LIN {X 0,Y 150.114,Z 268.264,A -85,B 0,C 180,E1 -24071.507,E2 -24071.507} C_VEL
LIN {X 0,Y 150.112,Z 268.281,A -85,B 0,C 180,E1 -24075.407,E2 -24075.407} C_VEL
LIN {X 0,Y 150.121,Z 268.245,A -85,B 0,C 180,E1 -24079.065,E2 -24079.065} C_VEL
LIN {X 0,Y 150.164,Z 268.273,A -85,B 0,C 180,E1 -24082.722,E2 -24082.722} C_VEL
LIN {X 0,Y 150.193,Z 268.249,A -85,B 0,C 180,E1 -24087.388,E2 -24087.388} C_VEL
LIN {X 0,Y 150.176,Z 268.244,A -85,B 0,C 180,E1 -24092.777,E2 -24092.777} C_VEL
LIN {X 0,Y 150.28,Z 268.247,A -85,B 0,C 180,E1 -24099.29,E2 -24099.29} C_VEL
LIN {X 0,Y 150.321,Z 268.203,A -85,B 0,C 180,E1 -24103.72,E2 -24103.72} C_VEL
LIN {X 0,Y 150.612,Z 268.222,A -85,B 0,C 180,E1 -24109.253,E2 -24109.253} C_VEL
LIN {X 0,Y 150.686,Z 268.205,A -85,B 0,C 180,E1 -24111.968,E2 -24111.968} C_VEL
LIN {X 0,Y 151.205,Z 268.124,A -85,B 0,C 180,E1 -24120.01,E2 -24120.01} C_VEL
LIN {X 0,Y 150.69,Z 268.169,A -85,B 0,C 180,E1 -24128.053,E2 -24128.053} C_VEL
LIN {X 0,Y 150.588,Z 268.188,A -85,B 0,C 180,E1 -24131.437,E2 -24131.437} C_VEL
LIN {X 0,Y 150.337,Z 268.255,A -85,B 0,C 180,E1 -24136.3,E2 -24136.3} C_VEL
LIN {X 0,Y 150.302,Z 268.224,A -85,B 0,C 180,E1 -24140.731,E2 -24140.731} C_VEL
LIN {X 0,Y 150.258,Z 268.254,A -85,B 0,C 180,E1 -24147.284,E2 -24147.284} C_VEL
LIN {X 0,Y 150.229,Z 268.268,A -85,B 0,C 180,E1 -24152.633,E2 -24152.633} C_VEL
LIN {X 0,Y 150.19,Z 268.256,A -85,B 0,C 180,E1 -24157.48,E2 -24157.48} C_VEL
LIN {X 0,Y 150.183,Z 268.457,A -85,B 0,C 180,E1 -24163.328,E2 -24163.328} C_VEL
LIN {X 0,Y 150.422,Z 269.542,A -85,B 0,C 180,E1 -24163.87,E2 -24163.87} C_VEL
LIN {X 0,Y 152.217,Z 272.467,A -85,B 0,C 180,E1 -24164.614,E2 -24164.614} C_VEL
LIN {X 0,Y 158.391,Z 283.05,A -85,B 0,C 180,E1 -24166.897,E2 -24166.897} C_VEL
LIN {X 0,Y 163.542,Z 294.743,A -85,B 0,C 180,E1 -24168.779,E2 -24168.779} C_VEL
LIN {X 0,Y 169.289,Z 310.581,A -85,B 0,C 180,E1 -24170.856,E2 -24170.856} C_VEL
LIN {X 0,Y 170.451,Z 314.297,A -85,B 0,C 180,E1 -24171.28,E2 -24171.28} C_VEL
LIN {X 0,Y 171.224,Z 322.163,A -85,B 0,C 180,E1 -24171.828,E2 -24171.828} C_VEL
LIN {X 0,Y 168.447,Z 373.925,A -85,B 0,C 180,E1 -24173.943,E2 -24173.943} C_VEL
LIN {X 0,Y 166.924,Z 387.276,A -85,B 0,C 180,E1 -24174.898,E2 -24174.898} C_VEL
LIN {X 0,Y 164.896,Z 400.456,A -85,B 0,C 180,E1 -24176.349,E2 -24176.349} C_VEL
LIN {X 0,Y 162.259,Z 413.148,A -85,B 0,C 180,E1 -24178.316,E2 -24178.316} C_VEL
LIN {X 0,Y 159.543,Z 424.472,A -85,B 0,C 180,E1 -24180.651,E2 -24180.651} C_VEL
LIN {X 0,Y 156.898,Z 434.655,A -85,B 0,C 180,E1 -24183.385,E2 -24183.385} C_VEL
LIN {X 0,Y 154.864,Z 442.186,A -85,B 0,C 180,E1 -24185.889,E2 -24185.889} C_VEL
LIN {X 0,Y 152.203,Z 451.403,A -85,B 0,C 180,E1 -24189.734,E2 -24189.734} C_VEL
LIN {X 0,Y 150.073,Z 458.797,A -85,B 0,C 180,E1 -24193.677,E2 -24193.677} C_VEL
LIN {X 0,Y 148.738,Z 464.717,A -85,B 0,C 180,E1 -24197.719,E2 -24197.719} C_VEL
LIN {X 0,Y 147.955,Z 469.35,A -85,B 0,C 180,E1 -24201.803,E2 -24201.803} C_VEL
LIN {X 0,Y 147.585,Z 472.609,A -85,B 0,C 180,E1 -24205.68,E2 -24205.68} C_VEL
LIN {X 0,Y 147.21,Z 473.67,A -85,B 0,C 180,E1 -24207.153,E2 -24207.153} C_VEL
LIN {X 0,Y 145.79,Z 474.919,A -85,B 0,C 180,E1 -24209.352,E2 -24209.352} C_VEL
LIN {X 0,Y 141.589,Z 476.74,A -85,B 0,C 180,E1 -24214.635,E2 -24214.635} C_VEL
LIN {X 0,Y 140.824,Z 477.165,A -85,B 0,C 180,E1 -24217.04,E2 -24217.04} C_VEL
LIN {X 0,Y 140.876,Z 477.218,A -85,B 0,C 180,E1 -24217.85,E2 -24217.85} C_VEL
LIN {X 0,Y 141.642,Z 477.292,A -85,B 0,C 180,E1 -24221.443,E2 -24221.443} C_VEL
LIN {X 0,Y 143.826,Z 476.121,A -85,B 0,C 180,E1 -24227.044,E2 -24227.044} C_VEL
LIN {X 0,Y 145.338,Z 474.921,A -85,B 0,C 180,E1 -24229.78,E2 -24229.78} C_VEL
LIN {X 0,Y 149.613,Z 471.328,A -85,B 0,C 180,E1 -24235.005,E2 -24235.005} C_VEL
LIN {X 0,Y 153.554,Z 467.474,A -85,B 0,C 180,E1 -24238.718,E2 -24238.718} C_VEL
LIN {X 0,Y 158.498,Z 462.018,A -85,B 0,C 180,E1 -24242.582,E2 -24242.582} C_VEL
LIN {X 0,Y 164.017,Z 455.204,A -85,B 0,C 180,E1 -24246.093,E2 -24246.093} C_VEL
LIN {X 0,Y 169.863,Z 447.238,A -85,B 0,C 180,E1 -24249.116,E2 -24249.116} C_VEL
LIN {X 0,Y 174.983,Z 439.159,A -85,B 0,C 180,E1 -24251.501,E2 -24251.501} C_VEL
LIN {X 0,Y 180.461,Z 429.331,A -85,B 0,C 180,E1 -24253.725,E2 -24253.725} C_VEL
LIN {X 0,Y 185.729,Z 418.252,A -85,B 0,C 180,E1 -24255.575,E2 -24255.575} C_VEL
LIN {X 0,Y 189.917,Z 407.478,A -85,B 0,C 180,E1 -24256.953,E2 -24256.953} C_VEL
LIN {X 0,Y 193.595,Z 395.64,A -85,B 0,C 180,E1 -24258.085,E2 -24258.085} C_VEL
LIN {X 0,Y 196.474,Z 383.38,A -85,B 0,C 180,E1 -24258.91,E2 -24258.91} C_VEL
LIN {X 0,Y 198.47,Z 370.195,A -85,B 0,C 180,E1 -24259.483,E2 -24259.483} C_VEL
LIN {X 0,Y 200.368,Z 346.995,A -85,B 0,C 180,E1 -24260.263,E2 -24260.263} C_VEL
LIN {X 0,Y 197.033,Z 338.865,A -85,B 0,C 180,E1 -24262.493,E2 -24262.493} C_VEL
LIN {X 0,Y 193.256,Z 330.702,A -85,B 0,C 180,E1 -24265.3,E2 -24265.3} C_VEL
LIN {X 0,Y 189.657,Z 323.776,A -85,B 0,C 180,E1 -24268.321,E2 -24268.321} C_VEL
LIN {X 0,Y 187.496,Z 319.855,A -85,B 0,C 180,E1 -24270.371,E2 -24270.371} C_VEL
LIN {X 0,Y 185.186,Z 315.819,A -85,B 0,C 180,E1 -24272.9,E2 -24272.9} C_VEL
LIN {X 0,Y 182.151,Z 310.78,A -85,B 0,C 180,E1 -24277.047,E2 -24277.047} C_VEL
LIN {X 0,Y 179.744,Z 308.026,A -85,B 0,C 180,E1 -24281.505,E2 -24281.505} C_VEL
LIN {X 0,Y 179.034,Z 305.82,A -85,B 0,C 180,E1 -24284.042,E2 -24284.042} C_VEL
LIN {X 0,Y 178.22,Z 305.34,A -85,B 0,C 180,E1 -24290.916,E2 -24290.916} C_VEL
LIN {X 0,Y 179.566,Z 306.018,A -85,B 0,C 180,E1 -24296.72,E2 -24296.72} C_VEL
LIN {X 0,Y 181.237,Z 309.585,A -85,B 0,C 180,E1 -24300.701,E2 -24300.701} C_VEL
LIN {X 0,Y 182.777,Z 311.232,A -85,B 0,C 180,E1 -24303.057,E2 -24303.057} C_VEL
LIN {X 0,Y 185.094,Z 314.817,A -85,B 0,C 180,E1 -24306.112,E2 -24306.112} C_VEL
LIN {X 0,Y 188.663,Z 320.369,A -85,B 0,C 180,E1 -24309.833,E2 -24309.833} C_VEL
LIN {X 0,Y 191.169,Z 324.419,A -85,B 0,C 180,E1 -24312.027,E2 -24312.027} C_VEL
LIN {X 0,Y 195.512,Z 332.715,A -85,B 0,C 180,E1 -24315.431,E2 -24315.431} C_VEL
LIN {X 0,Y 199.029,Z 340.465,A -85,B 0,C 180,E1 -24317.868,E2 -24317.868} C_VEL
LIN {X 0,Y 200.576,Z 344.145,A -85,B 0,C 180,E1 -24318.87,E2 -24318.87} C_VEL
LIN {X 0,Y 198.251,Z 370.487,A -85,B 0,C 180,E1 -24319.738,E2 -24319.738} C_VEL
LIN {X 0,Y 196.016,Z 383.546,A -85,B 0,C 180,E1 -24320.4,E2 -24320.4} C_VEL
LIN {X 0,Y 192.712,Z 396.803,A -85,B 0,C 180,E1 -24321.426,E2 -24321.426} C_VEL
LIN {X 0,Y 188.637,Z 408.974,A -85,B 0,C 180,E1 -24322.774,E2 -24322.774} C_VEL
LIN {X 0,Y 183.992,Z 420.098,A -85,B 0,C 180,E1 -24324.416,E2 -24324.416} C_VEL
LIN {X 0,Y 178.638,Z 430.756,A -85,B 0,C 180,E1 -24326.496,E2 -24326.496} C_VEL
LIN {X 0,Y 173.399,Z 439.603,A -85,B 0,C 180,E1 -24328.761,E2 -24328.761} C_VEL
LIN {X 0,Y 167.326,Z 448.476,A -85,B 0,C 180,E1 -24331.738,E2 -24331.738} C_VEL
LIN {X 0,Y 161.32,Z 456.16,A -85,B 0,C 180,E1 -24335.236,E2 -24335.236} C_VEL
LIN {X 0,Y 155.806,Z 462.351,A -85,B 0,C 180,E1 -24339.146,E2 -24339.146} C_VEL
LIN {X 0,Y 150.792,Z 467.378,A -85,B 0,C 180,E1 -24343.66,E2 -24343.66} C_VEL
LIN {X 0,Y 147.025,Z 470.599,A -85,B 0,C 180,E1 -24347.999,E2 -24347.999} C_VEL
LIN {X 0,Y 145.053,Z 472.047,A -85,B 0,C 180,E1 -24350.966,E2 -24350.966} C_VEL
LIN {X 0,Y 143.38,Z 473.04,A -85,B 0,C 180,E1 -24353.976,E2 -24353.976} C_VEL
LIN {X 0,Y 141.957,Z 473.566,A -85,B 0,C 180,E1 -24357.289,E2 -24357.289} C_VEL
LIN {X 0,Y 141.05,Z 473.582,A -85,B 0,C 180,E1 -24360.12,E2 -24360.12} C_VEL
LIN {X 0,Y 140.258,Z 472.896,A -85,B 0,C 180,E1 -24364.384,E2 -24364.384} C_VEL
LIN {X 0,Y 139.92,Z 470.954,A -85,B 0,C 180,E1 -24369.42,E2 -24369.42} C_VEL
LIN {X 0,Y 140.27,Z 468.071,A -85,B 0,C 180,E1 -24374.009,E2 -24374.009} C_VEL
LIN {X 0,Y 141.079,Z 464.088,A -85,B 0,C 180,E1 -24378.511,E2 -24378.511} C_VEL
LIN {X 0,Y 142.418,Z 458.667,A -85,B 0,C 180,E1 -24383.104,E2 -24383.104} C_VEL
LIN {X 0,Y 144.081,Z 452.41,A -85,B 0,C 180,E1 -24387.208,E2 -24387.208} C_VEL
LIN {X 0,Y 146.493,Z 444.212,A -85,B 0,C 180,E1 -24391.379,E2 -24391.379} C_VEL
LIN {X 0,Y 149.079,Z 435.528,A -85,B 0,C 180,E1 -24394.848,E2 -24394.848} C_VEL
LIN {X 0,Y 151.995,Z 425.557,A -85,B 0,C 180,E1 -24397.978,E2 -24397.978} C_VEL
LIN {X 0,Y 154.727,Z 415.315,A -85,B 0,C 180,E1 -24400.472,E2 -24400.472} C_VEL
LIN {X 0,Y 157.223,Z 404.192,A -85,B 0,C 180,E1 -24402.591,E2 -24402.591} C_VEL
LIN {X 0,Y 159.59,Z 391.565,A -85,B 0,C 180,E1 -24404.391,E2 -24404.391} C_VEL
LIN {X 0,Y 161.357,Z 378.639,A -85,B 0,C 180,E1 -24405.681,E2 -24405.681} C_VEL
LIN {X 0,Y 162.596,Z 365.189,A -85,B 0,C 180,E1 -24406.513,E2 -24406.513} C_VEL
LIN {X 0,Y 165.409,Z 315.499,A -85,B 0,C 180,E1 -24408.539,E2 -24408.539} C_VEL
LIN {X 0,Y 162.201,Z 305.506,A -85,B 0,C 180,E1 -24409.784,E2 -24409.784} C_VEL
LIN {X 0,Y 158.295,Z 296.088,A -85,B 0,C 180,E1 -24411.227,E2 -24411.227} C_VEL
LIN {X 0,Y 152.717,Z 285.561,A -85,B 0,C 180,E1 -24413.29,E2 -24413.29} C_VEL
LIN {X 0,Y 147.299,Z 276.795,A -85,B 0,C 180,E1 -24415.411,E2 -24415.411} C_VEL
LIN {X 0,Y 144.943,Z 272.955,A -85,B 0,C 180,E1 -24416.406,E2 -24416.406} C_VEL
LIN {X 0,Y 143.419,Z 270.299,A -85,B 0,C 180,E1 -24417.141,E2 -24417.141} C_VEL
LIN {X 0,Y 143.154,Z 269.269,A -85,B 0,C 180,E1 -24417.807,E2 -24417.807} C_VEL
LIN {X 0,Y 143.114,Z 269.139,A -85,B 0,C 180,E1 -24423.425,E2 -24423.425} C_VEL
LIN {X 0,Y 143.032,Z 269.137,A -85,B 0,C 180,E1 -24429.705,E2 -24429.705} C_VEL
LIN {X 0,Y 143.017,Z 269.169,A -85,B 0,C 180,E1 -24433.476,E2 -24433.476} C_VEL
LIN {X 0,Y 143.022,Z 269.135,A -85,B 0,C 180,E1 -24437.49,E2 -24437.49} C_VEL
LIN {X 0,Y 143.059,Z 269.144,A -85,B 0,C 180,E1 -24441.822,E2 -24441.822} C_VEL
LIN {X 0,Y 143.161,Z 269.123,A -85,B 0,C 180,E1 -24447.33,E2 -24447.33} C_VEL
LIN {X 0,Y 143.1,Z 269.139,A -85,B 0,C 180,E1 -24453.781,E2 -24453.781} C_VEL
LIN {X 0,Y 143.245,Z 269.11,A -85,B 0,C 180,E1 -24459.926,E2 -24459.926} C_VEL
LIN {X 0,Y 143.315,Z 269.092,A -85,B 0,C 180,E1 -24465.819,E2 -24465.819} C_VEL
LIN {X 0,Y 143.538,Z 269.101,A -85,B 0,C 180,E1 -24468.717,E2 -24468.717} C_VEL
LIN {X 0,Y 143.612,Z 269.088,A -85,B 0,C 180,E1 -24471.569,E2 -24471.569} C_VEL
LIN {X 0,Y 144.163,Z 268.998,A -85,B 0,C 180,E1 -24480.011,E2 -24480.011} C_VEL
LIN {X 0,Y 143.617,Z 269.046,A -85,B 0,C 180,E1 -24488.453,E2 -24488.453} C_VEL
LIN {X 0,Y 143.513,Z 269.069,A -85,B 0,C 180,E1 -24491.625,E2 -24491.625} C_VEL
LIN {X 0,Y 143.275,Z 269.126,A -85,B 0,C 180,E1 -24497.127,E2 -24497.127} C_VEL
LIN {X 0,Y 143.24,Z 269.103,A -85,B 0,C 180,E1 -24501.205,E2 -24501.205} C_VEL
LIN {X 0,Y 143.203,Z 269.124,A -85,B 0,C 180,E1 -24507.937,E2 -24507.937} C_VEL
LIN {X 0,Y 143.18,Z 269.151,A -85,B 0,C 180,E1 -24513.435,E2 -24513.435} C_VEL
LIN {X 0,Y 143.073,Z 269.163,A -85,B 0,C 180,E1 -24519.699,E2 -24519.699} C_VEL
LIN {X 0,Y 143.19,Z 269.508,A -85,B 0,C 180,E1 -24521.286,E2 -24521.286} C_VEL
LIN {X 0,Y 143.576,Z 270.92,A -85,B 0,C 180,E1 -24521.81,E2 -24521.81} C_VEL
LIN {X 0,Y 145.199,Z 273.4,A -85,B 0,C 180,E1 -24522.532,E2 -24522.532} C_VEL
LIN {X 0,Y 152.145,Z 284.806,A -85,B 0,C 180,E1 -24525.335,E2 -24525.335} C_VEL
LIN {X 0,Y 156.518,Z 294.087,A -85,B 0,C 180,E1 -24527.045,E2 -24527.045} C_VEL
LIN {X 0,Y 163.069,Z 311.701,A -85,B 0,C 180,E1 -24529.575,E2 -24529.575} C_VEL
LIN {X 0,Y 164.54,Z 316.772,A -85,B 0,C 180,E1 -24530.171,E2 -24530.171} C_VEL
LIN {X 0,Y 165.072,Z 323.799,A -85,B 0,C 180,E1 -24530.654,E2 -24530.654} C_VEL
LIN {X 0,Y 162.232,Z 373.888,A -85,B 0,C 180,E1 -24532.757,E2 -24532.757} C_VEL
LIN {X 0,Y 160.687,Z 386.922,A -85,B 0,C 180,E1 -24533.709,E2 -24533.709} C_VEL
LIN {X 0,Y 158.591,Z 400.189,A -85,B 0,C 180,E1 -24535.206,E2 -24535.206} C_VEL
LIN {X 0,Y 155.845,Z 412.921,A -85,B 0,C 180,E1 -24537.233,E2 -24537.233} C_VEL
LIN {X 0,Y 153.008,Z 424.268,A -85,B 0,C 180,E1 -24539.647,E2 -24539.647} C_VEL
LIN {X 0,Y 150.557,Z 433.462,A -85,B 0,C 180,E1 -24542.169,E2 -24542.169} C_VEL
LIN {X 0,Y 148.326,Z 441.116,A -85,B 0,C 180,E1 -24544.754,E2 -24544.754} C_VEL
LIN {X 0,Y 145.888,Z 449.142,A -85,B 0,C 180,E1 -24548.073,E2 -24548.073} C_VEL
LIN {X 0,Y 143.605,Z 456.961,A -85,B 0,C 180,E1 -24552.185,E2 -24552.185} C_VEL
LIN {X 0,Y 141.774,Z 464.124,A -85,B 0,C 180,E1 -24557.106,E2 -24557.106} C_VEL
LIN {X 0,Y 140.902,Z 468.867,A -85,B 0,C 180,E1 -24561.39,E2 -24561.39} C_VEL
LIN {X 0,Y 140.504,Z 472.459,A -85,B 0,C 180,E1 -24565.693,E2 -24565.693} C_VEL
LIN {X 0,Y 140.552,Z 475.017,A -85,B 0,C 180,E1 -24569.996,E2 -24569.996} C_VEL
LIN {X 0,Y 140.501,Z 476.202,A -85,B 0,C 180,E1 -24572.863,E2 -24572.863} C_VEL
LIN {X 0,Y 140.876,Z 477.218,A -85,B 0,C 180,E1 -24577.85,E2 -24577.85} C_VEL
LIN {X 0,Y 140.711,Z 477.362,A -85,B 0,C 180,E1 -24580.248,E2 -24580.248} C_VEL
LIN {X 0,Y 139.03,Z 476.948,A -85,B 0,C 180,E1 -24584.245,E2 -24584.245} C_VEL
LIN {X 0,Y 137.961,Z 476.22,A -85,B 0,C 180,E1 -24587.499,E2 -24587.499} C_VEL
LIN {X 0,Y 138.224,Z 475.379,A -85,B 0,C 180,E1 -24589.936,E2 -24589.936} C_VEL
LIN {X 0,Y 138.631,Z 475.043,A -85,B 0,C 180,E1 -24590.728,E2 -24590.728} C_VEL
LIN {X 0,Y 140.776,Z 473.481,A -85,B 0,C 180,E1 -24593.535,E2 -24593.535} C_VEL
LIN {X 0,Y 144.554,Z 470.408,A -85,B 0,C 180,E1 -24597.503,E2 -24597.503} C_VEL
LIN {X 0,Y 149.937,Z 465.259,A -85,B 0,C 180,E1 -24602.081,E2 -24602.081} C_VEL
LIN {X 0,Y 155.553,Z 459.12,A -85,B 0,C 180,E1 -24605.964,E2 -24605.964} C_VEL
LIN {X 0,Y 161.367,Z 452.117,A -85,B 0,C 180,E1 -24609.157,E2 -24609.157} C_VEL
LIN {X 0,Y 167.626,Z 443.425,A -85,B 0,C 180,E1 -24612.125,E2 -24612.125} C_VEL
LIN {X 0,Y 173.193,Z 434.55,A -85,B 0,C 180,E1 -24614.421,E2 -24614.421} C_VEL
LIN {X 0,Y 178.478,Z 424.816,A -85,B 0,C 180,E1 -24616.344,E2 -24616.344} C_VEL
LIN {X 0,Y 183.362,Z 414.102,A -85,B 0,C 180,E1 -24617.949,E2 -24617.949} C_VEL
LIN {X 0,Y 187.727,Z 402.178,A -85,B 0,C 180,E1 -24619.292,E2 -24619.292} C_VEL
LIN {X 0,Y 191.228,Z 389.812,A -85,B 0,C 180,E1 -24620.303,E2 -24620.303} C_VEL
LIN {X 0,Y 193.868,Z 376.677,A -85,B 0,C 180,E1 -24621.01,E2 -24621.01} C_VEL
LIN {X 0,Y 195.663,Z 360.309,A -85,B 0,C 180,E1 -24621.574,E2 -24621.574} C_VEL
LIN {X 0,Y 196.434,Z 349.811,A -85,B 0,C 180,E1 -24621.971,E2 -24621.971} C_VEL
LIN {X 0,Y 192.818,Z 340.819,A -85,B 0,C 180,E1 -24624.69,E2 -24624.69} C_VEL
LIN {X 0,Y 189.522,Z 333.784,A -85,B 0,C 180,E1 -24627.432,E2 -24627.432} C_VEL
LIN {X 0,Y 186.138,Z 326.946,A -85,B 0,C 180,E1 -24630.683,E2 -24630.683} C_VEL
LIN {X 0,Y 183.474,Z 322.178,A -85,B 0,C 180,E1 -24633.757,E2 -24633.757} C_VEL
LIN {X 0,Y 180.812,Z 317.581,A -85,B 0,C 180,E1 -24637.638,E2 -24637.638} C_VEL
LIN {X 0,Y 178.585,Z 314.736,A -85,B 0,C 180,E1 -24642.15,E2 -24642.15} C_VEL
LIN {X 0,Y 177.992,Z 312.818,A -85,B 0,C 180,E1 -24644.484,E2 -24644.484} C_VEL
LIN {X 0,Y 177.426,Z 312.457,A -85,B 0,C 180,E1 -24651.973,E2 -24651.973} C_VEL
LIN {X 0,Y 178.516,Z 313.044,A -85,B 0,C 180,E1 -24656.371,E2 -24656.371} C_VEL
LIN {X 0,Y 180.192,Z 316.644,A -85,B 0,C 180,E1 -24660.526,E2 -24660.526} C_VEL
LIN {X 0,Y 181.408,Z 317.944,A -85,B 0,C 180,E1 -24662.457,E2 -24662.457} C_VEL
LIN {X 0,Y 184.101,Z 322.429,A -85,B 0,C 180,E1 -24666.145,E2 -24666.145} C_VEL
LIN {X 0,Y 186.957,Z 327.052,A -85,B 0,C 180,E1 -24669.228,E2 -24669.228} C_VEL
LIN {X 0,Y 189.22,Z 330.907,A -85,B 0,C 180,E1 -24671.312,E2 -24671.312} C_VEL
LIN {X 0,Y 193.082,Z 338.646,A -85,B 0,C 180,E1 -24674.517,E2 -24674.517} C_VEL
LIN {X 0,Y 196.752,Z 347.3,A -85,B 0,C 180,E1 -24677.239,E2 -24677.239} C_VEL
LIN {X 0,Y 194.427,Z 371.29,A -85,B 0,C 180,E1 -24678,E2 -24678} C_VEL
LIN {X 0,Y 192.02,Z 384.641,A -85,B 0,C 180,E1 -24678.692,E2 -24678.692} C_VEL
LIN {X 0,Y 188.844,Z 396.794,A -85,B 0,C 180,E1 -24679.629,E2 -24679.629} C_VEL
LIN {X 0,Y 185.117,Z 407.735,A -85,B 0,C 180,E1 -24680.8,E2 -24680.8} C_VEL
LIN {X 0,Y 180.112,Z 419.458,A -85,B 0,C 180,E1 -24682.475,E2 -24682.475} C_VEL
LIN {X 0,Y 174.705,Z 429.992,A -85,B 0,C 180,E1 -24684.483,E2 -24684.483} C_VEL
LIN {X 0,Y 169.309,Z 438.891,A -85,B 0,C 180,E1 -24686.704,E2 -24686.704} C_VEL
LIN {X 0,Y 163.393,Z 447.266,A -85,B 0,C 180,E1 -24689.432,E2 -24689.432} C_VEL
LIN {X 0,Y 157.977,Z 454.009,A -85,B 0,C 180,E1 -24692.308,E2 -24692.308} C_VEL
LIN {X 0,Y 152.109,Z 460.521,A -85,B 0,C 180,E1 -24696.052,E2 -24696.052} C_VEL
LIN {X 0,Y 146.941,Z 465.572,A -85,B 0,C 180,E1 -24700.077,E2 -24700.077} C_VEL
LIN {X 0,Y 143.623,Z 468.426,A -85,B 0,C 180,E1 -24703.224,E2 -24703.224} C_VEL
LIN {X 0,Y 141.273,Z 470.276,A -85,B 0,C 180,E1 -24705.863,E2 -24705.863} C_VEL
LIN {X 0,Y 138.686,Z 472.074,A -85,B 0,C 180,E1 -24709.456,E2 -24709.456} C_VEL
LIN {X 0,Y 135.582,Z 473.575,A -85,B 0,C 180,E1 -24715.242,E2 -24715.242} C_VEL
LIN {X 0,Y 134.38,Z 473.729,A -85,B 0,C 180,E1 -24718.473,E2 -24718.473} C_VEL
LIN {X 0,Y 133.222,Z 473,A -85,B 0,C 180,E1 -24723.712,E2 -24723.712} C_VEL
LIN {X 0,Y 132.853,Z 471.42,A -85,B 0,C 180,E1 -24728.271,E2 -24728.271} C_VEL
LIN {X 0,Y 132.957,Z 469.404,A -85,B 0,C 180,E1 -24732.031,E2 -24732.031} C_VEL
LIN {X 0,Y 133.523,Z 466.275,A -85,B 0,C 180,E1 -24736.304,E2 -24736.304} C_VEL
LIN {X 0,Y 134.594,Z 461.695,A -85,B 0,C 180,E1 -24740.992,E2 -24740.992} C_VEL
LIN {X 0,Y 136.087,Z 455.876,A -85,B 0,C 180,E1 -24745.562,E2 -24745.562} C_VEL
LIN {X 0,Y 138.273,Z 448.545,A -85,B 0,C 180,E1 -24750.005,E2 -24750.005} C_VEL
LIN {X 0,Y 141.13,Z 439.696,A -85,B 0,C 180,E1 -24754.141,E2 -24754.141} C_VEL
LIN {X 0,Y 144.121,Z 429.904,A -85,B 0,C 180,E1 -24757.711,E2 -24757.711} C_VEL
LIN {X 0,Y 147.182,Z 419.302,A -85,B 0,C 180,E1 -24760.667,E2 -24760.667} C_VEL
LIN {X 0,Y 150.149,Z 407.524,A -85,B 0,C 180,E1 -24763.194,E2 -24763.194} C_VEL
LIN {X 0,Y 152.639,Z 395.551,A -85,B 0,C 180,E1 -24765.116,E2 -24765.116} C_VEL
LIN {X 0,Y 154.745,Z 382.299,A -85,B 0,C 180,E1 -24766.631,E2 -24766.631} C_VEL
LIN {X 0,Y 156.204,Z 369.079,A -85,B 0,C 180,E1 -24767.618,E2 -24767.618} C_VEL
LIN {X 0,Y 159.33,Z 316.877,A -85,B 0,C 180,E1 -24769.831,E2 -24769.831} C_VEL
LIN {X 0,Y 156.021,Z 306.942,A -85,B 0,C 180,E1 -24771.182,E2 -24771.182} C_VEL
LIN {X 0,Y 152.754,Z 299.02,A -85,B 0,C 180,E1 -24772.485,E2 -24772.485} C_VEL
LIN {X 0,Y 146.687,Z 287.801,A -85,B 0,C 180,E1 -24774.903,E2 -24774.903} C_VEL
LIN {X 0,Y 140.206,Z 277.357,A -85,B 0,C 180,E1 -24777.716,E2 -24777.716} C_VEL
LIN {X 0,Y 138.412,Z 274.513,A -85,B 0,C 180,E1 -24778.559,E2 -24778.559} C_VEL
LIN {X 0,Y 136.591,Z 272.017,A -85,B 0,C 180,E1 -24779.419,E2 -24779.419} C_VEL
LIN {X 0,Y 136.139,Z 270.606,A -85,B 0,C 180,E1 -24779.878,E2 -24779.878} C_VEL
LIN {X 0,Y 136.04,Z 270.074,A -85,B 0,C 180,E1 -24780.761,E2 -24780.761} C_VEL
LIN {X 0,Y 136.019,Z 270.031,A -85,B 0,C 180,E1 -24784.641,E2 -24784.641} C_VEL
LIN {X 0,Y 136.004,Z 270.013,A -85,B 0,C 180,E1 -24789.205,E2 -24789.205} C_VEL
LIN {X 0,Y 135.962,Z 270.049,A -85,B 0,C 180,E1 -24793.66,E2 -24793.66} C_VEL
LIN {X 0,Y 135.967,Z 270.01,A -85,B 0,C 180,E1 -24797.799,E2 -24797.799} C_VEL
LIN {X 0,Y 136.007,Z 270.018,A -85,B 0,C 180,E1 -24801.694,E2 -24801.694} C_VEL
LIN {X 0,Y 136.041,Z 270.032,A -85,B 0,C 180,E1 -24805.756,E2 -24805.756} C_VEL
LIN {X 0,Y 136.077,Z 269.99,A -85,B 0,C 180,E1 -24812.315,E2 -24812.315} C_VEL
LIN {X 0,Y 136.179,Z 270.006,A -85,B 0,C 180,E1 -24818.836,E2 -24818.836} C_VEL
LIN {X 0,Y 136.231,Z 269.962,A -85,B 0,C 180,E1 -24825.064,E2 -24825.064} C_VEL
LIN {X 0,Y 136.43,Z 269.981,A -85,B 0,C 180,E1 -24828.19,E2 -24828.19} C_VEL
LIN {X 0,Y 136.541,Z 269.972,A -85,B 0,C 180,E1 -24831.129,E2 -24831.129} C_VEL
LIN {X 0,Y 137.12,Z 269.872,A -85,B 0,C 180,E1 -24840.011,E2 -24840.011} C_VEL
LIN {X 0,Y 136.547,Z 269.923,A -85,B 0,C 180,E1 -24848.894,E2 -24848.894} C_VEL
LIN {X 0,Y 136.429,Z 269.952,A -85,B 0,C 180,E1 -24851.903,E2 -24851.903} C_VEL
LIN {X 0,Y 136.186,Z 269.995,A -85,B 0,C 180,E1 -24858.049,E2 -24858.049} C_VEL
LIN {X 0,Y 136.166,Z 269.985,A -85,B 0,C 180,E1 -24861.703,E2 -24861.703} C_VEL
LIN {X 0,Y 136.112,Z 270.001,A -85,B 0,C 180,E1 -24868.616,E2 -24868.616} C_VEL
LIN {X 0,Y 136.089,Z 270.022,A -85,B 0,C 180,E1 -24874.628,E2 -24874.628} C_VEL
LIN {X 0,Y 136.089,Z 270.288,A -85,B 0,C 180,E1 -24878.693,E2 -24878.693} C_VEL
LIN {X 0,Y 136.325,Z 271.367,A -85,B 0,C 180,E1 -24879.243,E2 -24879.243} C_VEL
LIN {X 0,Y 137.833,Z 273.901,A -85,B 0,C 180,E1 -24880.018,E2 -24880.018} C_VEL
LIN {X 0,Y 139.072,Z 275.551,A -85,B 0,C 180,E1 -24880.581,E2 -24880.581} C_VEL
LIN {X 0,Y 145.984,Z 286.748,A -85,B 0,C 180,E1 -24883.641,E2 -24883.641} C_VEL
LIN {X 0,Y 149.605,Z 293.741,A -85,B 0,C 180,E1 -24885.156,E2 -24885.156} C_VEL
LIN {X 0,Y 154.655,Z 306.593,A -85,B 0,C 180,E1 -24887.283,E2 -24887.283} C_VEL
LIN {X 0,Y 158.573,Z 318.303,A -85,B 0,C 180,E1 -24888.902,E2 -24888.902} C_VEL
LIN {X 0,Y 159.04,Z 324.789,A -85,B 0,C 180,E1 -24889.366,E2 -24889.366} C_VEL
LIN {X 0,Y 156.01,Z 374.531,A -85,B 0,C 180,E1 -24891.516,E2 -24891.516} C_VEL
LIN {X 0,Y 154.434,Z 387.339,A -85,B 0,C 180,E1 -24892.502,E2 -24892.502} C_VEL
LIN {X 0,Y 152.354,Z 399.917,A -85,B 0,C 180,E1 -24893.969,E2 -24893.969} C_VEL
LIN {X 0,Y 149.912,Z 411.106,A -85,B 0,C 180,E1 -24895.762,E2 -24895.762} C_VEL
LIN {X 0,Y 147.629,Z 420.142,A -85,B 0,C 180,E1 -24897.613,E2 -24897.613} C_VEL
LIN {X 0,Y 144.917,Z 430.026,A -85,B 0,C 180,E1 -24900.188,E2 -24900.188} C_VEL
LIN {X 0,Y 141.803,Z 440.027,A -85,B 0,C 180,E1 -24903.504,E2 -24903.504} C_VEL
LIN {X 0,Y 139.776,Z 446.724,A -85,B 0,C 180,E1 -24906.277,E2 -24906.277} C_VEL
LIN {X 0,Y 137.191,Z 455.007,A -85,B 0,C 180,E1 -24910.546,E2 -24910.546} C_VEL
LIN {X 0,Y 135.326,Z 461.655,A -85,B 0,C 180,E1 -24914.945,E2 -24914.945} C_VEL
LIN {X 0,Y 134.125,Z 466.923,A -85,B 0,C 180,E1 -24919.428,E2 -24919.428} C_VEL
LIN {X 0,Y 133.531,Z 470.986,A -85,B 0,C 180,E1 -24923.953,E2 -24923.953} C_VEL
LIN {X 0,Y 133.417,Z 473.076,A -85,B 0,C 180,E1 -24926.976,E2 -24926.976} C_VEL
LIN {X 0,Y 133.471,Z 474.722,A -85,B 0,C 180,E1 -24929.995,E2 -24929.995} C_VEL
LIN {X 0,Y 133.416,Z 475.951,A -85,B 0,C 180,E1 -24933.015,E2 -24933.015} C_VEL
LIN {X 0,Y 133.807,Z 477.057,A -85,B 0,C 180,E1 -24938.067,E2 -24938.067} C_VEL
LIN {X 0,Y 134.664,Z 477.214,A -85,B 0,C 180,E1 -24942.045,E2 -24942.045} C_VEL
LIN {X 0,Y 137.018,Z 476.145,A -85,B 0,C 180,E1 -24947.919,E2 -24947.919} C_VEL
LIN {X 0,Y 138.631,Z 475.043,A -85,B 0,C 180,E1 -24950.728,E2 -24950.728} C_VEL
LIN {X 0,Y 139.631,Z 474,A -85,B 0,C 180,E1 -24953.094,E2 -24953.094} C_VEL
LIN {X 0,Y 140.142,Z 471.75,A -85,B 0,C 180,E1 -24957.052,E2 -24957.052} C_VEL
LIN {X 0,Y 141.25,Z 468.717,A -85,B 0,C 180,E1 -24960.871,E2 -24960.871} C_VEL
LIN {X 0,Y 143.12,Z 466.45,A -85,B 0,C 180,E1 -24962.938,E2 -24962.938} C_VEL
LIN {X 0,Y 148.068,Z 461.595,A -85,B 0,C 180,E1 -24966.386,E2 -24966.386} C_VEL
LIN {X 0,Y 153.832,Z 455.221,A -85,B 0,C 180,E1 -24969.757,E2 -24969.757} C_VEL
LIN {X 0,Y 160.277,Z 447.292,A -85,B 0,C 180,E1 -24972.811,E2 -24972.811} C_VEL
LIN {X 0,Y 165.88,Z 439.258,A -85,B 0,C 180,E1 -24975.202,E2 -24975.202} C_VEL
LIN {X 0,Y 171.814,Z 429.484,A -85,B 0,C 180,E1 -24977.41,E2 -24977.41} C_VEL
LIN {X 0,Y 177.48,Z 418.513,A -85,B 0,C 180,E1 -24979.223,E2 -24979.223} C_VEL
LIN {X 0,Y 182.589,Z 406.116,A -85,B 0,C 180,E1 -24980.765,E2 -24980.765} C_VEL
LIN {X 0,Y 186.517,Z 393.956,A -85,B 0,C 180,E1 -24981.861,E2 -24981.861} C_VEL
LIN {X 0,Y 189.678,Z 380.376,A -85,B 0,C 180,E1 -24982.682,E2 -24982.682} C_VEL
LIN {X 0,Y 191.638,Z 366.976,A -85,B 0,C 180,E1 -24983.184,E2 -24983.184} C_VEL
LIN {X 0,Y 192.789,Z 352.895,A -85,B 0,C 180,E1 -24983.691,E2 -24983.691} C_VEL
LIN {X 0,Y 189.257,Z 343.942,A -85,B 0,C 180,E1 -24986.647,E2 -24986.647} C_VEL
LIN {X 0,Y 185.849,Z 336.533,A -85,B 0,C 180,E1 -24989.852,E2 -24989.852} C_VEL
LIN {X 0,Y 183.68,Z 332.203,A -85,B 0,C 180,E1 -24992.221,E2 -24992.221} C_VEL
LIN {X 0,Y 181.679,Z 328.274,A -85,B 0,C 180,E1 -24994.808,E2 -24994.808} C_VEL
LIN {X 0,Y 179.646,Z 324.488,A -85,B 0,C 180,E1 -24997.996,E2 -24997.996} C_VEL
LIN {X 0,Y 177.52,Z 321.651,A -85,B 0,C 180,E1 -25002.555,E2 -25002.555} C_VEL
LIN {X 0,Y 176.991,Z 319.827,A -85,B 0,C 180,E1 -25004.817,E2 -25004.817} C_VEL
LIN {X 0,Y 176.397,Z 319.429,A -85,B 0,C 180,E1 -25010.821,E2 -25010.821} C_VEL
LIN {X 0,Y 177.472,Z 320.069,A -85,B 0,C 180,E1 -25016.018,E2 -25016.018} C_VEL
LIN {X 0,Y 179.153,Z 323.675,A -85,B 0,C 180,E1 -25020.35,E2 -25020.35} C_VEL
LIN {X 0,Y 180.218,Z 325.049,A -85,B 0,C 180,E1 -25022.131,E2 -25022.131} C_VEL
LIN {X 0,Y 182.55,Z 329.042,A -85,B 0,C 180,E1 -25025.476,E2 -25025.476} C_VEL
LIN {X 0,Y 185.284,Z 333.689,A -85,B 0,C 180,E1 -25028.615,E2 -25028.615} C_VEL
LIN {X 0,Y 187.173,Z 337.132,A -85,B 0,C 180,E1 -25030.462,E2 -25030.462} C_VEL
LIN {X 0,Y 190.763,Z 344.671,A -85,B 0,C 180,E1 -25033.626,E2 -25033.626} C_VEL
LIN {X 0,Y 193.016,Z 350.388,A -85,B 0,C 180,E1 -25035.467,E2 -25035.467} C_VEL
LIN {X 0,Y 190.977,Z 371.158,A -85,B 0,C 180,E1 -25036.16,E2 -25036.16} C_VEL
LIN {X 0,Y 188.583,Z 384.082,A -85,B 0,C 180,E1 -25036.801,E2 -25036.801} C_VEL
LIN {X 0,Y 185.418,Z 396.075,A -85,B 0,C 180,E1 -25037.706,E2 -25037.706} C_VEL
LIN {X 0,Y 181.129,Z 408.207,A -85,B 0,C 180,E1 -25038.967,E2 -25038.967} C_VEL
LIN {X 0,Y 176.321,Z 419.123,A -85,B 0,C 180,E1 -25040.512,E2 -25040.512} C_VEL
LIN {X 0,Y 170.342,Z 430.332,A -85,B 0,C 180,E1 -25042.62,E2 -25042.62} C_VEL
LIN {X 0,Y 164.614,Z 439.338,A -85,B 0,C 180,E1 -25044.883,E2 -25044.883} C_VEL
LIN {X 0,Y 158.541,Z 447.515,A -85,B 0,C 180,E1 -25047.563,E2 -25047.563} C_VEL
LIN {X 0,Y 153.113,Z 453.941,A -85,B 0,C 180,E1 -25050.312,E2 -25050.312} C_VEL
LIN {X 0,Y 147.634,Z 459.737,A -85,B 0,C 180,E1 -25053.592,E2 -25053.592} C_VEL
LIN {X 0,Y 142.015,Z 464.977,A -85,B 0,C 180,E1 -25057.653,E2 -25057.653} C_VEL
LIN {X 0,Y 137.647,Z 468.556,A -85,B 0,C 180,E1 -25061.57,E2 -25061.57} C_VEL
LIN {X 0,Y 133.204,Z 471.65,A -85,B 0,C 180,E1 -25066.701,E2 -25066.701} C_VEL
LIN {X 0,Y 131.038,Z 472.853,A -85,B 0,C 180,E1 -25069.946,E2 -25069.946} C_VEL
LIN {X 0,Y 128.401,Z 473.773,A -85,B 0,C 180,E1 -25075.163,E2 -25075.163} C_VEL
LIN {X 0,Y 126.792,Z 473.63,A -85,B 0,C 180,E1 -25080.081,E2 -25080.081} C_VEL
LIN {X 0,Y 126.16,Z 472.953,A -85,B 0,C 180,E1 -25083.541,E2 -25083.541} C_VEL
LIN {X 0,Y 125.788,Z 471.852,A -85,B 0,C 180,E1 -25086.983,E2 -25086.983} C_VEL
LIN {X 0,Y 125.817,Z 469.547,A -85,B 0,C 180,E1 -25091.685,E2 -25091.685} C_VEL
LIN {X 0,Y 126.555,Z 465.67,A -85,B 0,C 180,E1 -25097.171,E2 -25097.171} C_VEL
LIN {X 0,Y 127.999,Z 460.013,A -85,B 0,C 180,E1 -25102.83,E2 -25102.83} C_VEL
LIN {X 0,Y 129.805,Z 453.608,A -85,B 0,C 180,E1 -25107.678,E2 -25107.678} C_VEL
LIN {X 0,Y 132.4,Z 445.714,A -85,B 0,C 180,E1 -25112.286,E2 -25112.286} C_VEL
LIN {X 0,Y 135.101,Z 437.585,A -85,B 0,C 180,E1 -25115.977,E2 -25115.977} C_VEL
LIN {X 0,Y 138.287,Z 427.634,A -85,B 0,C 180,E1 -25119.512,E2 -25119.512} C_VEL
LIN {X 0,Y 141.585,Z 416.528,A -85,B 0,C 180,E1 -25122.547,E2 -25122.547} C_VEL
LIN {X 0,Y 144.305,Z 405.655,A -85,B 0,C 180,E1 -25124.819,E2 -25124.819} C_VEL
LIN {X 0,Y 146.825,Z 393.686,A -85,B 0,C 180,E1 -25126.695,E2 -25126.695} C_VEL
LIN {X 0,Y 148.843,Z 380.888,A -85,B 0,C 180,E1 -25128.144,E2 -25128.144} C_VEL
LIN {X 0,Y 150.214,Z 368.642,A -85,B 0,C 180,E1 -25129.033,E2 -25129.033} C_VEL
LIN {X 0,Y 153.343,Z 318.463,A -85,B 0,C 180,E1 -25131.2,E2 -25131.2} C_VEL
LIN {X 0,Y 149.453,Z 307.002,A -85,B 0,C 180,E1 -25132.912,E2 -25132.912} C_VEL
LIN {X 0,Y 144.878,Z 297.438,A -85,B 0,C 180,E1 -25134.846,E2 -25134.846} C_VEL
LIN {X 0,Y 138.826,Z 286.828,A -85,B 0,C 180,E1 -25137.545,E2 -25137.545} C_VEL
LIN {X 0,Y 134.177,Z 279.582,A -85,B 0,C 180,E1 -25139.777,E2 -25139.777} C_VEL
LIN {X 0,Y 131.421,Z 275.439,A -85,B 0,C 180,E1 -25141.197,E2 -25141.197} C_VEL
LIN {X 0,Y 129.557,Z 273.048,A -85,B 0,C 180,E1 -25142.185,E2 -25142.185} C_VEL
LIN {X 0,Y 129.041,Z 271.474,A -85,B 0,C 180,E1 -25142.766,E2 -25142.766} C_VEL
LIN {X 0,Y 128.974,Z 270.956,A -85,B 0,C 180,E1 -25143.555,E2 -25143.555} C_VEL
LIN {X 0,Y 128.915,Z 270.894,A -85,B 0,C 180,E1 -25150.272,E2 -25150.272} C_VEL
LIN {X 0,Y 128.896,Z 270.922,A -85,B 0,C 180,E1 -25155.145,E2 -25155.145} C_VEL
LIN {X 0,Y 128.92,Z 270.883,A -85,B 0,C 180,E1 -25159.754,E2 -25159.754} C_VEL
LIN {X 0,Y 128.945,Z 270.922,A -85,B 0,C 180,E1 -25164.849,E2 -25164.849} C_VEL
LIN {X 0,Y 128.973,Z 270.863,A -85,B 0,C 180,E1 -25170.686,E2 -25170.686} C_VEL
LIN {X 0,Y 129.065,Z 270.903,A -85,B 0,C 180,E1 -25177.787,E2 -25177.787} C_VEL
LIN {X 0,Y 129.151,Z 270.836,A -85,B 0,C 180,E1 -25184.225,E2 -25184.225} C_VEL
LIN {X 0,Y 129.348,Z 270.86,A -85,B 0,C 180,E1 -25187.983,E2 -25187.983} C_VEL
LIN {X 0,Y 129.466,Z 270.856,A -85,B 0,C 180,E1 -25190.64,E2 -25190.64} C_VEL
LIN {X 0,Y 130.075,Z 270.746,A -85,B 0,C 180,E1 -25200.012,E2 -25200.012} C_VEL
LIN {X 0,Y 129.473,Z 270.802,A -85,B 0,C 180,E1 -25209.384,E2 -25209.384} C_VEL
LIN {X 0,Y 129.313,Z 270.845,A -85,B 0,C 180,E1 -25212.568,E2 -25212.568} C_VEL
LIN {X 0,Y 129.102,Z 270.865,A -85,B 0,C 180,E1 -25219.076,E2 -25219.076} C_VEL
LIN {X 0,Y 129.063,Z 270.874,A -85,B 0,C 180,E1 -25222.419,E2 -25222.419} C_VEL
LIN {X 0,Y 129.022,Z 270.912,A -85,B 0,C 180,E1 -25225.847,E2 -25225.847} C_VEL
LIN {X 0,Y 129.038,Z 270.879,A -85,B 0,C 180,E1 -25229.365,E2 -25229.365} C_VEL
LIN {X 0,Y 129.014,Z 271.01,A -85,B 0,C 180,E1 -25235.528,E2 -25235.528} C_VEL
LIN {X 0,Y 129.16,Z 271.911,A -85,B 0,C 180,E1 -25236.3,E2 -25236.3} C_VEL
LIN {X 0,Y 130.653,Z 274.711,A -85,B 0,C 180,E1 -25237.253,E2 -25237.253} C_VEL
LIN {X 0,Y 131.959,Z 276.06,A -85,B 0,C 180,E1 -25237.903,E2 -25237.903} C_VEL
LIN {X 0,Y 134.058,Z 279.441,A -85,B 0,C 180,E1 -25238.997,E2 -25238.997} C_VEL
LIN {X 0,Y 139.553,Z 288.182,A -85,B 0,C 180,E1 -25241.629,E2 -25241.629} C_VEL
LIN {X 0,Y 143.807,Z 295.875,A -85,B 0,C 180,E1 -25243.546,E2 -25243.546} C_VEL
LIN {X 0,Y 148.377,Z 307.33,A -85,B 0,C 180,E1 -25245.635,E2 -25245.635} C_VEL
LIN {X 0,Y 152.684,Z 320.262,A -85,B 0,C 180,E1 -25247.566,E2 -25247.566} C_VEL
LIN {X 0,Y 153.105,Z 324.998,A -85,B 0,C 180,E1 -25247.947,E2 -25247.947} C_VEL
LIN {X 0,Y 150.004,Z 374.066,A -85,B 0,C 180,E1 -25250.107,E2 -25250.107} C_VEL
LIN {X 0,Y 148.36,Z 386.99,A -85,B 0,C 180,E1 -25251.117,E2 -25251.117} C_VEL
LIN {X 0,Y 146.187,Z 399.639,A -85,B 0,C 180,E1 -25252.626,E2 -25252.626} C_VEL
LIN {X 0,Y 143.649,Z 410.881,A -85,B 0,C 180,E1 -25254.475,E2 -25254.475} C_VEL
LIN {X 0,Y 141.244,Z 419.93,A -85,B 0,C 180,E1 -25256.384,E2 -25256.384} C_VEL
LIN {X 0,Y 138.407,Z 429.84,A -85,B 0,C 180,E1 -25259.056,E2 -25259.056} C_VEL
LIN {X 0,Y 135.392,Z 438.944,A -85,B 0,C 180,E1 -25262.144,E2 -25262.144} C_VEL
LIN {X 0,Y 133.288,Z 445.811,A -85,B 0,C 180,E1 -25265.045,E2 -25265.045} C_VEL
LIN {X 0,Y 130.494,Z 454.236,A -85,B 0,C 180,E1 -25269.504,E2 -25269.504} C_VEL
LIN {X 0,Y 128.442,Z 461.004,A -85,B 0,C 180,E1 -25274.117,E2 -25274.117} C_VEL
LIN {X 0,Y 127.143,Z 466.386,A -85,B 0,C 180,E1 -25278.84,E2 -25278.84} C_VEL
LIN {X 0,Y 126.465,Z 470.551,A -85,B 0,C 180,E1 -25283.614,E2 -25283.614} C_VEL
LIN {X 0,Y 126.326,Z 472.733,A -85,B 0,C 180,E1 -25286.806,E2 -25286.806} C_VEL
LIN {X 0,Y 126.382,Z 474.427,A -85,B 0,C 180,E1 -25289.995,E2 -25289.995} C_VEL
LIN {X 0,Y 126.325,Z 475.699,A -85,B 0,C 180,E1 -25293.184,E2 -25293.184} C_VEL
LIN {X 0,Y 126.972,Z 477.066,A -85,B 0,C 180,E1 -25299.553,E2 -25299.553} C_VEL
LIN {X 0,Y 128.812,Z 476.836,A -85,B 0,C 180,E1 -25305.826,E2 -25305.826} C_VEL
LIN {X 0,Y 132.035,Z 475.116,A -85,B 0,C 180,E1 -25311.871,E2 -25311.871} C_VEL
LIN {X 0,Y 134.288,Z 473.644,A -85,B 0,C 180,E1 -25314.746,E2 -25314.746} C_VEL
LIN {X 0,Y 138.288,Z 470.671,A -85,B 0,C 180,E1 -25318.863,E2 -25318.863} C_VEL
LIN {X 0,Y 143.12,Z 466.45,A -85,B 0,C 180,E1 -25322.938,E2 -25322.938} C_VEL
LIN {X 0,Y 145.13,Z 464.066,A -85,B 0,C 180,E1 -25324.927,E2 -25324.927} C_VEL
LIN {X 0,Y 147.228,Z 459.904,A -85,B 0,C 180,E1 -25328.366,E2 -25328.366} C_VEL
LIN {X 0,Y 149.64,Z 455.19,A -85,B 0,C 180,E1 -25331.588,E2 -25331.588} C_VEL
LIN {X 0,Y 152.037,Z 451.846,A -85,B 0,C 180,E1 -25333.187,E2 -25333.187} C_VEL
LIN {X 0,Y 158.654,Z 443.511,A -85,B 0,C 180,E1 -25336.035,E2 -25336.035} C_VEL
LIN {X 0,Y 164.664,Z 434.719,A -85,B 0,C 180,E1 -25338.318,E2 -25338.318} C_VEL
LIN {X 0,Y 170.399,Z 425.066,A -85,B 0,C 180,E1 -25340.184,E2 -25340.184} C_VEL
LIN {X 0,Y 175.604,Z 414.532,A -85,B 0,C 180,E1 -25341.754,E2 -25341.754} C_VEL
LIN {X 0,Y 180.28,Z 402.795,A -85,B 0,C 180,E1 -25343.044,E2 -25343.044} C_VEL
LIN {X 0,Y 184.093,Z 390.376,A -85,B 0,C 180,E1 -25344.038,E2 -25344.038} C_VEL
LIN {X 0,Y 186.927,Z 377.588,A -85,B 0,C 180,E1 -25344.723,E2 -25344.723} C_VEL
LIN {X 0,Y 188.76,Z 363.04,A -85,B 0,C 180,E1 -25345.223,E2 -25345.223} C_VEL
LIN {X 0,Y 189.319,Z 356.174,A -85,B 0,C 180,E1 -25345.486,E2 -25345.486} C_VEL
LIN {X 0,Y 186.401,Z 348.489,A -85,B 0,C 180,E1 -25348.181,E2 -25348.181} C_VEL
LIN {X 0,Y 183.35,Z 341.575,A -85,B 0,C 180,E1 -25351.355,E2 -25351.355} C_VEL
LIN {X 0,Y 181.693,Z 338.02,A -85,B 0,C 180,E1 -25353.398,E2 -25353.398} C_VEL
LIN {X 0,Y 180.106,Z 334.709,A -85,B 0,C 180,E1 -25355.633,E2 -25355.633} C_VEL
LIN {X 0,Y 178.291,Z 331.219,A -85,B 0,C 180,E1 -25358.69,E2 -25358.69} C_VEL
LIN {X 0,Y 176.316,Z 328.15,A -85,B 0,C 180,E1 -25363.524,E2 -25363.524} C_VEL
LIN {X 0,Y 175.996,Z 326.837,A -85,B 0,C 180,E1 -25365.153,E2 -25365.153} C_VEL
LIN {X 0,Y 175.487,Z 326.471,A -85,B 0,C 180,E1 -25370.773,E2 -25370.773} C_VEL
LIN {X 0,Y 176.425,Z 327.047,A -85,B 0,C 180,E1 -25375.613,E2 -25375.613} C_VEL
LIN {X 0,Y 178.114,Z 330.713,A -85,B 0,C 180,E1 -25380.172,E2 -25380.172} C_VEL
LIN {X 0,Y 178.907,Z 331.856,A -85,B 0,C 180,E1 -25381.572,E2 -25381.572} C_VEL
LIN {X 0,Y 180.945,Z 335.484,A -85,B 0,C 180,E1 -25384.682,E2 -25384.682} C_VEL
LIN {X 0,Y 183.467,Z 340.024,A -85,B 0,C 180,E1 -25387.794,E2 -25387.794} C_VEL
LIN {X 0,Y 185.625,Z 344.269,A -85,B 0,C 180,E1 -25390.043,E2 -25390.043} C_VEL
LIN {X 0,Y 188.529,Z 350.927,A -85,B 0,C 180,E1 -25392.762,E2 -25392.762} C_VEL
LIN {X 0,Y 189.563,Z 353.696,A -85,B 0,C 180,E1 -25393.681,E2 -25393.681} C_VEL
LIN {X 0,Y 187.424,Z 373.176,A -85,B 0,C 180,E1 -25394.328,E2 -25394.328} C_VEL
LIN {X 0,Y 184.924,Z 385.675,A -85,B 0,C 180,E1 -25394.972,E2 -25394.972} C_VEL
LIN {X 0,Y 181.336,Z 398.131,A -85,B 0,C 180,E1 -25395.929,E2 -25395.929} C_VEL
LIN {X 0,Y 176.629,Z 410.529,A -85,B 0,C 180,E1 -25397.277,E2 -25397.277} C_VEL
LIN {X 0,Y 171.669,Z 421.001,A -85,B 0,C 180,E1 -25398.8,E2 -25398.8} C_VEL
LIN {X 0,Y 166.133,Z 430.774,A -85,B 0,C 180,E1 -25400.673,E2 -25400.673} C_VEL
LIN {X 0,Y 160.211,Z 439.642,A -85,B 0,C 180,E1 -25402.908,E2 -25402.908} C_VEL
LIN {X 0,Y 153.869,Z 447.764,A -85,B 0,C 180,E1 -25405.577,E2 -25405.577} C_VEL
LIN {X 0,Y 146.973,Z 455.452,A -85,B 0,C 180,E1 -25408.995,E2 -25408.995} C_VEL
LIN {X 0,Y 141.352,Z 460.912,A -85,B 0,C 180,E1 -25412.312,E2 -25412.312} C_VEL
LIN {X 0,Y 135.513,Z 465.916,A -85,B 0,C 180,E1 -25416.508,E2 -25416.508} C_VEL
LIN {X 0,Y 130.48,Z 469.61,A -85,B 0,C 180,E1 -25421.063,E2 -25421.063} C_VEL
LIN {X 0,Y 125.945,Z 472.321,A -85,B 0,C 180,E1 -25426.484,E2 -25426.484} C_VEL
LIN {X 0,Y 123.072,Z 473.554,A -85,B 0,C 180,E1 -25431.093,E2 -25431.093} C_VEL
LIN {X 0,Y 121.413,Z 473.907,A -85,B 0,C 180,E1 -25434.637,E2 -25434.637} C_VEL
LIN {X 0,Y 120.134,Z 473.826,A -85,B 0,C 180,E1 -25438.237,E2 -25438.237} C_VEL
LIN {X 0,Y 119.265,Z 473.206,A -85,B 0,C 180,E1 -25442.086,E2 -25442.086} C_VEL
LIN {X 0,Y 118.793,Z 472.227,A -85,B 0,C 180,E1 -25445.541,E2 -25445.541} C_VEL
LIN {X 0,Y 118.688,Z 469.677,A -85,B 0,C 180,E1 -25451.291,E2 -25451.291} C_VEL
LIN {X 0,Y 119.289,Z 466.359,A -85,B 0,C 180,E1 -25456.375,E2 -25456.375} C_VEL
LIN {X 0,Y 120.604,Z 461.322,A -85,B 0,C 180,E1 -25462.046,E2 -25462.046} C_VEL
LIN {X 0,Y 122.532,Z 454.738,A -85,B 0,C 180,E1 -25467.54,E2 -25467.54} C_VEL
LIN {X 0,Y 125.029,Z 447.098,A -85,B 0,C 180,E1 -25472.421,E2 -25472.421} C_VEL
LIN {X 0,Y 127.889,Z 439.245,A -85,B 0,C 180,E1 -25476.315,E2 -25476.315} C_VEL
LIN {X 0,Y 131.097,Z 429.71,A -85,B 0,C 180,E1 -25480.039,E2 -25480.039} C_VEL
LIN {X 0,Y 134.48,Z 419.017,A -85,B 0,C 180,E1 -25483.222,E2 -25483.222} C_VEL
LIN {X 0,Y 137.734,Z 407.136,A -85,B 0,C 180,E1 -25485.923,E2 -25485.923} C_VEL
LIN {X 0,Y 140.502,Z 394.787,A -85,B 0,C 180,E1 -25487.978,E2 -25487.978} C_VEL
LIN {X 0,Y 142.76,Z 381.317,A -85,B 0,C 180,E1 -25489.574,E2 -25489.574} C_VEL
LIN {X 0,Y 144.178,Z 369.345,A -85,B 0,C 180,E1 -25490.489,E2 -25490.489} C_VEL
LIN {X 0,Y 147.476,Z 319.921,A -85,B 0,C 180,E1 -25492.679,E2 -25492.679} C_VEL
LIN {X 0,Y 143.343,Z 308.294,A -85,B 0,C 180,E1 -25494.623,E2 -25494.623} C_VEL
LIN {X 0,Y 137.961,Z 297.656,A -85,B 0,C 180,E1 -25497.092,E2 -25497.092} C_VEL
LIN {X 0,Y 131.575,Z 286.895,A -85,B 0,C 180,E1 -25500.256,E2 -25500.256} C_VEL
LIN {X 0,Y 127.368,Z 280.614,A -85,B 0,C 180,E1 -25502.539,E2 -25502.539} C_VEL
LIN {X 0,Y 125.182,Z 277.266,A -85,B 0,C 180,E1 -25503.832,E2 -25503.832} C_VEL
LIN {X 0,Y 124.308,Z 276.246,A -85,B 0,C 180,E1 -25504.343,E2 -25504.343} C_VEL
LIN {X 0,Y 122.515,Z 273.935,A -85,B 0,C 180,E1 -25505.447,E2 -25505.447} C_VEL
LIN {X 0,Y 121.97,Z 272.381,A -85,B 0,C 180,E1 -25506.079,E2 -25506.079} C_VEL
LIN {X 0,Y 121.842,Z 271.833,A -85,B 0,C 180,E1 -25507.194,E2 -25507.194} C_VEL
LIN {X 0,Y 121.845,Z 271.779,A -85,B 0,C 180,E1 -25511.446,E2 -25511.446} C_VEL
LIN {X 0,Y 121.832,Z 271.764,A -85,B 0,C 180,E1 -25518.591,E2 -25518.591} C_VEL
LIN {X 0,Y 121.897,Z 271.8,A -85,B 0,C 180,E1 -25524.809,E2 -25524.809} C_VEL
LIN {X 0,Y 121.895,Z 271.743,A -85,B 0,C 180,E1 -25529.874,E2 -25529.874} C_VEL
LIN {X 0,Y 121.976,Z 271.789,A -85,B 0,C 180,E1 -25537.215,E2 -25537.215} C_VEL
LIN {X 0,Y 122.062,Z 271.714,A -85,B 0,C 180,E1 -25543.283,E2 -25543.283} C_VEL
LIN {X 0,Y 122.291,Z 271.732,A -85,B 0,C 180,E1 -25547.705,E2 -25547.705} C_VEL
LIN {X 0,Y 122.395,Z 271.738,A -85,B 0,C 180,E1 -25550.094,E2 -25550.094} C_VEL
LIN {X 0,Y 122.561,Z 271.652,A -85,B 0,C 180,E1 -25556.726,E2 -25556.726} C_VEL
LIN {X 0,Y 123.029,Z 271.621,A -85,B 0,C 180,E1 -25560.013,E2 -25560.013} C_VEL
LIN {X 0,Y 122.413,Z 271.698,A -85,B 0,C 180,E1 -25566.606,E2 -25566.606} C_VEL
